ELSIF Device.bFirstCycle THEN
	(* first call of the server device since reboot/reset *)
	bReady := FALSE;
	_PresentValue_Priority12 := BACnetBinaryPV_NULL;
ELSE
	(* server device not ready, reset local ready also *)
	bReady := FALSE;
	nErrorId := nERR_OPERATIONAL;
END_IF
(* set error flag *)
bError := (nErrorId <> nERR_NO_ERROR);
END_FUNCTION_BLOCK

(* POU FB_BACnet_BinaryOutput_ADS, ST *)
FUNCTION_BLOCK FB_BACnet_BinaryOutput_ADS
VAR_INPUT
	bEnablePV		: BOOL;
	bPV				: BOOL; (* present value bool type *)
	bManual			: BOOL; (* FALSE --> TRUE: write present_value immediately, FALSE: only write present_value on-change, TRUE: write present_value on-change and when device turns operational *)
	ePriority		: E_BACNETPRIORITY := BACNETPRIORITY_12;
END_VAR
VAR_IN_OUT
	Device			: FB_BACnet_Device;
END_VAR
VAR_OUTPUT
	bReady			: BOOL;
	bPvDone			: BOOL; (* present_value written over ADS *)
	bPresentValue	: BOOL;
	bOverridden		: BOOL;
	bOutOfService	: BOOL;
	bFault			: BOOL;
	bInAlarm		: BOOL;
	bError			: BOOL;
	nErrorId		: UINT;
	nAdsErrorId		: UDINT;
END_VAR
VAR
	_PresentValue AT%I*: WORD; 			(* ~(BACnet_PresentValue 			:		: )
								   			(BACnet_ObjectType 				: BO	: )	*)
    _PresentValue_Ads : WORD;
	_StatusFlags AT%I*: WORD; 			(* ~(BACnet_StatusFlags 			:		: )	*)
	_ObjectId AT%I*: DWORD;				(* ~(BACnet_ObjectIdentifier			 :		: LINK) *)
	_StatusFlagsBits : ST_BACnet_StatusFlags;
	_nUpdateCount : UDINT := 0;
	_WriteProp : FB_BACnet_WriteProp;
	_rtrigManual : R_TRIG;
	_bEnPvOld : BOOL;
	_nObjType : E_BACNETOBJECTTYPE;
END_VAR
VAR CONSTANT
	nERR_NO_ERROR		: UINT := 0;
	nERR_WRONG_MAPPING	: UINT := 2;
	nERR_OPERATIONAL	: UINT := 3;
	nERR_WRONG_TYPE		: UINT := 4;
END_VAR
(* update server device *)
IF Device._nUpdateCount = _nUpdateCount THEN
	Device();
END_IF
(* remind current number of update counter *)
_nUpdateCount := Device._nUpdateCount;

(* trigger on manual flag *)
_rtrigManual(CLK:= bManual, Q=> );

(* decode object type *)
_nObjType := F_BACnet_GetObjType(_ObjectId);

(* check BitString format of StatusFlags --> if StatusFlags are less than 4, object isn't linked correctly *)
IF _nObjType <> BACnetObjectType_BinaryOutput THEN
	(* wrong mapped object type *)
	nErrorId := nERR_WRONG_TYPE;
	bReady := FALSE;
	bPvDone := FALSE;

ELSIF (_StatusFlags < 4) THEN
	(* wrong mapping *)
	nErrorId := nERR_WRONG_MAPPING;
	bReady := FALSE;
	bPvDone := FALSE;

ELSIF Device.bOperational THEN
	(* write present_value on manual trigger, on-change and on operational recover *)
	IF		_rtrigManual.Q
		OR	((F_BACnet_IsFinite(_PresentValue_Ads) <> F_BACnet_IsFinite(_PresentValue_Ads)) AND bEnablePV)
		OR	(bPV <> F_BinPV_To_Bool(_PresentValue_Ads) AND bEnablePV)
		OR	((NOT bReady) AND bManual)
		OR	(bEnablePV <> _bEnPvOld)
	THEN
		_WriteProp.bExecute := TRUE;
		bPvDone := FALSE;
		(* write depending on enable state *)
		_PresentValue_Ads := F_Bool_To_BinPV(bEnablePV, bPV);
		_bEnPvOld := bEnablePV;
	END_IF

	(* ready state *)
	bReady := TRUE;
	nErrorId := nERR_NO_ERROR;


	(* present value *)
	bPresentValue := F_BinPV_To_Bool(_PresentValue);

	(* build bit states *)
	_StatusFlagsBits := F_BACnet_StatusFlags(_StatusFlags);

	(* copy states to output *)
	bOverridden := _StatusFlagsBits.overridden;
	bOutOfService := _StatusFlagsBits.out_of_service;
	bFault := _StatusFlagsBits.fault;
	bInAlarm := _StatusFlagsBits.in_alarm;

ELSIF Device.bFirstCycle THEN
	(* first call of the server device since reboot/reset *)
	bReady := FALSE;
	bPvDone := FALSE;
ELSE
	(* server device not ready, reset local ready also *)
	bReady := FALSE;
	nErrorId := nERR_OPERATIONAL;
	bPvDone := FALSE;
END_IF

(* call write property command *)
_WriteProp(
	BACnetDevicePort	:= Device.nAdsPort,
	bExecute			:= ,
	sNetId				:= Device.sAmsNetId,
	ObjectType			:= _nObjType,
	PropertyID			:= BACnetPropertyIdentifier_PresentValue,
	Priority			:= ePriority,
	DataType			:= BACnetDataType_BinaryPV,
	ObjectInstance		:= F_BACnet_GetObjInstance(_ObjectId),
	ptrValue			:= ADR(_PresentValue_Ads),
	nLenValue			:= SIZEOF(_PresentValue_Ads),
	bDone				=> ,
	bBusy				=> ,
	bError				=> ,
	nErrID				=> nAdsErrorId);

(* set done flag *)
IF _WriteProp.bExecute AND (NOT _WriteProp.bBusy) THEN
	(* reset execution bit *)
	_WriteProp(bExecute := FALSE);
	(* check if command was finished with error *)
	IF _WriteProp.bError THEN
		IF bManual THEN
			(* retrigger if manual flag is set *)
			_WriteProp.bExecute := TRUE;
		END_IF
		bPvDone := FALSE;
	ELSE
		(* successful written *)
		bPvDone	:= TRUE;
	END_IF
END_IF

(* set error flag *)
bError := (nErrorId <> nERR_NO_ERROR) OR (nAdsErrorId <> 0);
END_FUNCTION_BLOCK

(* POU FB_BACnet_BinaryOutput_EX, ST *)
FUNCTION_BLOCK FB_BACnet_BinaryOutput_EX
VAR_INPUT
	bEnablePV	: BOOL; (* enable present value with priority x in priority array, FALSE = priority x disable (NULL) *)
	bPV			: BOOL; (* present value bool type *)
END_VAR
VAR_IN_OUT
	Device		: FB_BACnet_Device;
END_VAR
VAR_OUTPUT
	bReady			: BOOL;
	bPresentValue	: BOOL;
	bOverridden		: BOOL;
	bOutOfService	: BOOL;
	bFault			: BOOL;
	bInAlarm		: BOOL;
	bNoOutput		: BOOL;
	bOpenLoop		: BOOL;
	bShortedLoop	: BOOL;
	bOtherFault		: BOOL;
	eEventState		: E_BACNETEVENTSTATE;
	bAckedTrans_ToOffNormal : BOOL;
	bAckedTrans_ToFault		: BOOL;
	bAckedTrans_ToNormal	: BOOL;
	nActivePrio		: UINT;
	bError			: BOOL;
	nErrorId		: UINT;
END_VAR
VAR_INPUT
END_VAR
VAR
	_PresentValue AT%I*: WORD; 			(* ~(BACnet_PresentValue 			:		: )
								   			(BACnet_ObjectType 				: BO	: )	*)
    _PresentValue_Priority12 AT%Q*: WORD;(* ~(BACnet_PresentValue_Priority12	:		: )	*)
	_StatusFlags AT%I*: WORD; 			(* ~(BACnet_StatusFlags 			:		: )	*)
	_StatusFlagsBits : ST_BACnet_StatusFlags;
	_EventState AT%I*: WORD; 			(* ~(BACnet_EventState 				:		: )	*)
	_Reliability AT%I*: WORD;			(* ~(BACnet_Reliability 			:		: )	*)
	_ActivePriority AT%I*: UDINT; 		(* ~(BACnet_ActivePriority 			:		: )	*)
	_AckedTransitions AT%I*:WORD;	(* ~(BACnet_AckedTransitions:		: ) *)
	_AckedTransBits : ST_BACnet_EventTransitionBits;
	_nUpdateCount : UDINT := 0;
END_VAR
VAR CONSTANT
	nERR_NO_ERROR		: UINT := 0;
	nERR_WRONG_MAPPING	: UINT := 2;
	nERR_OPERATIONAL	: UINT := 3;
END_VAR
(* update server device *)
IF Device._nUpdateCount = _nUpdateCount THEN
	Device();
END_IF
(* remind current number of update counter *)
_nUpdateCount := Device._nUpdateCount;

(* check BitString format of StatusFlags --> if StatusFlags are less than 4, object isn't linked correctly *)
IF (_StatusFlags < 4) OR _AckedTransitions < 5 THEN
	(* wrong mapping *)
	nErrorId := nERR_WRONG_MAPPING;
	bReady := FALSE;

ELSIF Device.bOperational THEN
	(* ready state *)
	bReady := TRUE;
	nErrorId := nERR_NO_ERROR;

	(* write into priority array *)
	_PresentValue_Priority12 := F_Bool_To_BinPV(bEnablePV, bPV);

	(* present value *)
	bPresentValue := F_BinPV_To_Bool(_PresentValue);

	(* build bit states *)
	_StatusFlagsBits := F_BACnet_StatusFlags(_StatusFlags);
	_AckedTransBits		:= F_BACnet_EventTransitionFlags(_AckedTransitions);

	(* copy states to output *)
	bOverridden := _StatusFlagsBits.overridden;
	bOutOfService := _StatusFlagsBits.out_of_service;
	bFault := _StatusFlagsBits.fault;
	bInAlarm := _StatusFlagsBits.in_alarm;
	bNoOutput := (_Reliability = BACnetReliability_no_output);
	bOpenLoop := (_Reliability = BACnetReliability_open_loop);
	bShortedLoop := (_Reliability = BACnetReliability_shorted_loop);
	bOtherFault := (_Reliability = BACnetReliability_unreliable_other);
	bAckedTrans_ToOffNormal := _AckedTransBits.to_offnormal;
	bAckedTrans_ToFault := _AckedTransBits.to_fault;
	bAckedTrans_ToNormal := _AckedTransBits.to_normal;

	(* convert enumeration *)
	eEventState := _EventState;

	(* copy active priority *)
	nActivePrio := UDINT_TO_UINT(_ActivePriority);
ELSIF Device.bFirstCycle THEN
	(* first call of the server device since reboot/reset *)
	bReady := FALSE;
	_PresentValue_Priority12 := BACnetBinaryPV_NULL;
ELSE
	(* server device not ready, reset local ready also *)
	bReady := FALSE;
	nErrorId := nERR_OPERATIONAL;
END_IF
(* set error flag *)
bError := (nErrorId <> nERR_NO_ERROR);
END_FUNCTION_BLOCK

(* POU FB_BACnet_BinaryOutput_RAW, ST *)
FUNCTION_BLOCK FB_BACnet_BinaryOutput_RAW
VAR_INPUT
	bEnablePV	: BOOL; (* enable present value with priority x in priority array, FALSE = priority x disable (NULL) *)
	bPV			: BOOL; (* present value bool type *)
END_VAR
VAR_IN_OUT
	Device		: FB_BACnet_Device;
END_VAR
VAR_OUTPUT
	bReady			: BOOL;
	bPresentValue	: BOOL;
	bOverridden		: BOOL;
	bOutOfService	: BOOL;
	bFault			: BOOL;
	bInAlarm		: BOOL;
	bAckedTrans_ToOffNormal : BOOL;
	bAckedTrans_ToFault		: BOOL;
	bAckedTrans_ToNormal	: BOOL;
	bError			: BOOL;
	nErrorId		: UINT;
	bRawOut			AT%I*: BOOL;(* ~(BACnet_RawIoBinaryBoolValue : : ) *)
END_VAR
VAR
	_PresentValue AT%I*: WORD; 			(* ~(BACnet_PresentValue 			:		: )
								   			(BACnet_ObjectType 				: BO	: )	*)
    _PresentValue_Priority12 AT%Q*: WORD;(* ~(BACnet_PresentValue_Priority12	:		: )	*)
	_StatusFlags AT%I*: WORD; 			(* ~(BACnet_StatusFlags 			:		: )	*)
	_AckedTransitions AT%I*:WORD;		(* ~(BACnet_AckedTransitions:		: ) *)
	_AckedTransBits : ST_BACnet_EventTransitionBits;
	_StatusFlagsBits : ST_BACnet_StatusFlags;
	_nUpdateCount : UDINT := 0;
END_VAR
VAR CONSTANT
	nERR_NO_ERROR		: UINT := 0;
	nERR_WRONG_MAPPING	: UINT := 2;
	nERR_OPERATIONAL	: UINT := 3;
END_VAR
(* update server device *)
IF Device._nUpdateCount = _nUpdateCount THEN
	Device();
END_IF
(* remind current number of update counter *)
_nUpdateCount := Device._nUpdateCount;

(* check BitString format of StatusFlags --> if StatusFlags are less than 4, object isn't linked correctly *)
IF (_StatusFlags < 4) OR _AckedTransitions < 5 THEN
	(* wrong mapping *)
	nErrorId := nERR_WRONG_MAPPING;
	bReady := FALSE;

ELSIF Device.bOperational THEN
	(* ready state *)
	bReady := TRUE;
	nErrorId := nERR_NO_ERROR;

	(* write into priority array *)
	_PresentValue_Priority12 := F_Bool_To_BinPV(bEnablePV, bPV);

	(* present value *)
	bPresentValue := F_BinPV_To_Bool(_PresentValue);

	(* build bit states *)
	_StatusFlagsBits := F_BACnet_StatusFlags(_StatusFlags);
	_AckedTransBits		:= F_BACnet_EventTransitionFlags(_AckedTransitions);

	(* copy states to output *)
	bOverridden := _StatusFlagsBits.overridden;
	bOutOfService := _StatusFlagsBits.out_of_service;
	bFault := _StatusFlagsBits.fault;
	bInAlarm := _StatusFlagsBits.in_alarm;
	bAckedTrans_ToOffNormal := _AckedTransBits.to_offnormal;
	bAckedTrans_ToFault := _AckedTransBits.to_fault;
	bAckedTrans_ToNormal := _AckedTransBits.to_normal;

ELSIF Device.bFirstCycle THEN
	(* first call of the server device since reboot/reset *)
	bReady := FALSE;
	_PresentValue_Priority12 := BACnetBinaryPV_NULL;
ELSE
	(* server device not ready, reset local ready also *)
	bReady := FALSE;
	nErrorId := nERR_OPERATIONAL;
END_IF
(* set error flag *)
bError := (nErrorId <> nERR_NO_ERROR);
END_FUNCTION_BLOCK

(* POU FB_BACnet_BinaryValue, ST *)
FUNCTION_BLOCK FB_BACnet_BinaryValue
VAR_INPUT
	bEnablePV	: BOOL; (* enable present value with priority x in priority array, FALSE = priority x disable (NULL) *)
	bPV			: BOOL; (* present value bool type *)
END_VAR
VAR_IN_OUT
	Device		: FB_BACnet_Device;
END_VAR
VAR_OUTPUT
	bReady			: BOOL;
	bPresentValue	: BOOL;
	bOverridden		: BOOL;
	bOutOfService	: BOOL;
	bFault			: BOOL;
	bInAlarm		: BOOL;
	bError			: BOOL;
	nErrorId		: UINT;
END_VAR
VAR
	_PresentValue AT%I*: WORD; 			(* ~(BACnet_PresentValue 			:		: )
								   			(BACnet_ObjectType 				: BV	: )	*)
    _PresentValue_Priority12 AT%Q*: WORD;(* ~(BACnet_PresentValue_Priority12	:		: )	*)
	_StatusFlags AT%I*: WORD; 			(* ~(BACnet_StatusFlags 			:		: )	*)
	_StatusFlagsBits : ST_BACnet_StatusFlags;
	_nUpdateCount : UDINT := 0;
END_VAR
VAR CONSTANT
	nERR_NO_ERROR		: UINT := 0;
	nERR_WRONG_MAPPING	: UINT := 2;
	nERR_OPERATIONAL	: UINT := 3;
END_VAR
(* update server device *)
IF Device._nUpdateCount = _nUpdateCount THEN
	Device();
END_IF
(* remind current number of update counter *)
_nUpdateCount := Device._nUpdateCount;

(* check BitString format of StatusFlags --> if StatusFlags are less than 4, object isn't linked correctly *)
IF (_StatusFlags < 4) THEN
	(* wrong mapping *)
	nErrorId := nERR_WRONG_MAPPING;
	bReady := FALSE;

ELSIF Device.bOperational THEN
	(* ready state *)
	bReady := TRUE;
	nErrorId := nERR_NO_ERROR;

	(* write into priority array *)
	_PresentValue_Priority12 := F_Bool_To_BinPV(bEnablePV, bPV);

	(* present value *)
	bPresentValue := F_BinPV_To_Bool(_PresentValue);

	(* build bit states *)
	_StatusFlagsBits := F_BACnet_StatusFlags(_StatusFlags);

	(* copy states to output *)
	bOverridden := _StatusFlagsBits.overridden;
	bOutOfService := _StatusFlagsBits.out_of_service;
	bFault := _StatusFlagsBits.fault;
	bInAlarm := _StatusFlagsBits.in_alarm;

ELSIF Device.bFirstCycle THEN
	(* first call of the server device since reboot/reset *)
	bReady := FALSE;
	_PresentValue_Priority12 := BACnetBinaryPV_NULL;
ELSE
	(* server device not ready, reset local ready also *)
	bReady := FALSE;
	nErrorId := nERR_OPERATIONAL;
END_IF
(* set error flag *)
bError := (nErrorId <> nERR_NO_ERROR);
END_FUNCTION_BLOCK

(* POU FB_BACnet_BinaryValue_ADS, ST *)
FUNCTION_BLOCK FB_BACnet_BinaryValue_ADS
VAR_INPUT
	bEnablePV		: BOOL;
	bPV				: BOOL; (* present value bool type *)
	bManual			: BOOL; (* FALSE --> TRUE: write present_value immediately, FALSE: only write present_value on-change, TRUE: write present_value on-change and when device turns operational *)
	ePriority		: E_BACNETPRIORITY := BACNETPRIORITY_12;
END_VAR
VAR_IN_OUT
	Device			: FB_BACnet_Device;
END_VAR
VAR_OUTPUT
	bReady			: BOOL;
	bPvDone			: BOOL; (* present_value written over ADS *)
	bPresentValue	: BOOL;
	bOverridden		: BOOL;
	bOutOfService	: BOOL;
	bFault			: BOOL;
	bInAlarm		: BOOL;
	bError			: BOOL;
	nErrorId		: UINT;
	nAdsErrorId		: UDINT;
END_VAR
VAR
	_PresentValue AT%I*: WORD; 			(* ~(BACnet_PresentValue 			:		: )
								   			(BACnet_ObjectType 				: BV	: )	*)
    _PresentValue_Ads : WORD;
	_StatusFlags AT%I*: WORD; 			(* ~(BACnet_StatusFlags 			:		: )	*)
	_ObjectId AT%I*: DWORD;				(* ~(BACnet_ObjectIdentifier			 :		: LINK) *)
	_StatusFlagsBits : ST_BACnet_StatusFlags;
	_nUpdateCount : UDINT := 0;
	_WriteProp : FB_BACnet_WriteProp;
	_rtrigManual : R_TRIG;
	_bEnPvOld : BOOL;
	_nObjType : E_BACNETOBJECTTYPE;
END_VAR
VAR CONSTANT
	nERR_NO_ERROR		: UINT := 0;
	nERR_WRONG_MAPPING	: UINT := 2;
	nERR_OPERATIONAL	: UINT := 3;
	nERR_WRONG_TYPE		: UINT := 4;
END_VAR
(* update server device *)
IF Device._nUpdateCount = _nUpdateCount THEN
	Device();
END_IF
(* remind current number of update counter *)
_nUpdateCount := Device._nUpdateCount;

(* trigger on manual flag *)
_rtrigManual(CLK:= bManual, Q=> );

(* decode object type *)
_nObjType := F_BACnet_GetObjType(_ObjectId);

(* check BitString format of StatusFlags --> if StatusFlags are less than 4, object isn't linked correctly *)
IF _nObjType <> BACnetObjectType_BinaryValue THEN
	(* wrong mapped object type *)
	nErrorId := nERR_WRONG_TYPE;
	bReady := FALSE;
	bPvDone := FALSE;

ELSIF (_StatusFlags < 4) THEN
	(* wrong mapping *)
	nErrorId := nERR_WRONG_MAPPING;
	bReady := FALSE;
	bPvDone := FALSE;

ELSIF Device.bOperational THEN
	(* write present_value on manual trigger, on-change and on operational recover *)
	IF		_rtrigManual.Q
		OR	((F_BACnet_IsFinite(_PresentValue_Ads) <> F_BACnet_IsFinite(_PresentValue_Ads)) AND bEnablePV)
		OR	(bPV <> F_BinPV_To_Bool(_PresentValue_Ads) AND bEnablePV)
		OR	((NOT bReady) AND bManual)
		OR	(bEnablePV <> _bEnPvOld)
	THEN
		_WriteProp.bExecute := TRUE;
		bPvDone := FALSE;
		(* write depending on enable state *)
		_PresentValue_Ads := F_Bool_To_BinPV(bEnablePV, bPV);
		_bEnPvOld := bEnablePV;
	END_IF

	(* ready state *)
	bReady := TRUE;
	nErrorId := nERR_NO_ERROR;

	(* present value *)
	bPresentValue := F_BinPV_To_Bool(_PresentValue);

	(* build bit states *)
	_StatusFlagsBits := F_BACnet_StatusFlags(_StatusFlags);

	(* copy states to output *)
	bOverridden := _StatusFlagsBits.overridden;
	bOutOfService := _StatusFlagsBits.out_of_service;
	bFault := _StatusFlagsBits.fault;
	bInAlarm := _StatusFlagsBits.in_alarm;

ELSIF Device.bFirstCycle THEN
	(* first call of the server device since reboot/reset *)
	bReady := FALSE;
	bPvDone := FALSE;
ELSE
	(* server device not ready, reset local ready also *)
	bReady := FALSE;
	nErrorId := nERR_OPERATIONAL;
	bPvDone := FALSE;
END_IF

(* call write property command *)
_WriteProp(
	BACnetDevicePort	:= Device.nAdsPort,
	bExecute			:= ,
	sNetId				:= Device.sAmsNetId,
	ObjectType			:= _nObjType,
	PropertyID			:= BACnetPropertyIdentifier_PresentValue,
	Priority			:= ePriority,
	DataType			:= BACnetDataType_BinaryPV,
	ObjectInstance		:= F_BACnet_GetObjInstance(_ObjectId),
	ptrValue			:= ADR(_PresentValue_Ads),
	nLenValue			:= SIZEOF(_PresentValue_Ads),
	bDone				=> ,
	bBusy				=> ,
	bError				=> ,
	nErrID				=> nAdsErrorId);

(* set done flag *)
IF _WriteProp.bExecute AND (NOT _WriteProp.bBusy) THEN
	(* reset execution bit *)
	_WriteProp(bExecute := FALSE);
	(* check if command was finished with error *)
	IF _WriteProp.bError THEN
		IF bManual THEN
			(* retrigger if manual flag is set *)
			_WriteProp.bExecute := TRUE;
		END_IF
		bPvDone := FALSE;
	ELSE
		(* successful written *)
		bPvDone	:= TRUE;
	END_IF
END_IF

(* set error flag *)
bError := (nErrorId <> nERR_NO_ERROR) OR (nAdsErrorId <> 0);
END_FUNCTION_BLOCK

(* POU FB_BACnet_BinaryValue_EX, ST *)
FUNCTION_BLOCK FB_BACnet_BinaryValue_EX
VAR_INPUT
	bEnablePV	: BOOL; (* enable present value with priority x in priority array, FALSE = priority x disable (NULL) *)
	bPV			: BOOL; (* present value bool type *)
END_VAR
VAR_IN_OUT
	Device		: FB_BACnet_Device;
END_VAR
VAR_OUTPUT
	bReady			: BOOL;
	bPresentValue	: BOOL;
	bOverridden		: BOOL;
	bOutOfService	: BOOL;
	bFault			: BOOL;
	bInAlarm		: BOOL;
	bOtherFault		: BOOL;
	eEventState		: E_BACNETEVENTSTATE;
	bAckedTrans_ToOffNormal : BOOL;
	bAckedTrans_ToFault		: BOOL;
	bAckedTrans_ToNormal	: BOOL;
	nActivePrio		: UINT;
	bError			: BOOL;
	nErrorId		: UINT;
END_VAR
VAR

	_PresentValue AT%I*: WORD; 			(* ~(BACnet_PresentValue 			:		: )
								   			(BACnet_ObjectType 				: BV	: )	*)
    _PresentValue_Priority12 AT%Q*: WORD;(* ~(BACnet_PresentValue_Priority12	:		: )	*)
	_StatusFlags AT%I*: WORD; 			(* ~(BACnet_StatusFlags 			:		: )	*)
	_StatusFlagsBits : ST_BACnet_StatusFlags;
	_EventState AT%I*: WORD; 			(* ~(BACnet_EventState 				:		: )	*)
	_Reliability AT%I*: WORD;			(* ~(BACnet_Reliability 			:		: )	*)
	_ActivePriority AT%I*: UDINT; 		(* ~(BACnet_ActivePriority 			:		: )	*)
	_AckedTransitions AT%I*:WORD;		(* ~(BACnet_AckedTransitions:		: ) *)
	_AckedTransBits : ST_BACnet_EventTransitionBits;
	_nUpdateCount : UDINT := 0;
END_VAR
VAR CONSTANT
	nERR_NO_ERROR		: UINT := 0;
	nERR_WRONG_MAPPING	: UINT := 2;
	nERR_OPERATIONAL	: UINT := 3;
END_VAR
(* update server device *)
IF Device._nUpdateCount = _nUpdateCount THEN
	Device();
END_IF
(* remind current number of update counter *)
_nUpdateCount := Device._nUpdateCount;

(* check BitString format of StatusFlags --> if StatusFlags are less than 4, object isn't linked correctly *)
IF (_StatusFlags < 4) OR _AckedTransitions < 5 THEN
	(* wrong mapping *)
	nErrorId := nERR_WRONG_MAPPING;
	bReady := FALSE;

ELSIF Device.bOperational THEN
	(* ready state *)
	bReady := TRUE;
	nErrorId := nERR_NO_ERROR;

	(* write into priority array *)
	_PresentValue_Priority12 := F_Bool_To_BinPV(bEnablePV, bPV);

	(* present value *)
	bPresentValue := F_BinPV_To_Bool(_PresentValue);

	(* build bit states *)
	_StatusFlagsBits := F_BACnet_StatusFlags(_StatusFlags);
	_AckedTransBits		:= F_BACnet_EventTransitionFlags(_AckedTransitions);

	(* copy states to output *)
	bOverridden := _StatusFlagsBits.overridden;
	bOutOfService := _StatusFlagsBits.out_of_service;
	bFault := _StatusFlagsBits.fault;
	bInAlarm := _StatusFlagsBits.in_alarm;
	bOtherFault := (_Reliability = BACnetReliability_unreliable_other);
	bAckedTrans_ToOffNormal := _AckedTransBits.to_offnormal;
	bAckedTrans_ToFault := _AckedTransBits.to_fault;
	bAckedTrans_ToNormal := _AckedTransBits.to_normal;

	(* convert enumeration *)
	eEventState := _EventState;

	(* copy active priority *)
	nActivePrio := UDINT_TO_UINT(_ActivePriority);
ELSIF Device.bFirstCycle THEN
	(* first call of the server device since reboot/reset *)
	bReady := FALSE;
	_PresentValue_Priority12 := BACnetBinaryPV_NULL;
ELSE
	(* server device not ready, reset local ready also *)
	bReady := FALSE;
	nErrorId := nERR_OPERATIONAL;
END_IF
(* set error flag *)
bError := (nErrorId <> nERR_NO_ERROR);
END_FUNCTION_BLOCK

(* POU FB_BACnet_Calendar, ST *)
FUNCTION_BLOCK FB_BACnet_Calendar
VAR_IN_OUT
	Device	: FB_BACnet_Device;
END_VAR
VAR_OUTPUT
	bReady			: BOOL;
	bPresentValue	: BOOL;
	bError			: BOOL;
	nErrorId		: UINT;
END_VAR
VAR
	_PresentValue AT%I*: BOOL;	(* ~(BACnet_PresentValue 				 :		: )
									(BACnet_ObjectType 					 : CAL	: )	*)
	_nUpdateCount : UDINT := 0;
END_VAR
VAR CONSTANT
	nERR_NO_ERROR		: UINT := 0;
	nERR_OPERATIONAL	: UINT := 3;
END_VAR
(* update server device *)
IF Device._nUpdateCount = _nUpdateCount THEN
	Device();
END_IF
(* remind current number of update counter *)
_nUpdateCount := Device._nUpdateCount;

IF Device.bOperational THEN
	(* ready state *)
	bReady := TRUE;
	nErrorId := nERR_NO_ERROR;
	(* present value *)
	bPresentValue := _PresentValue;
ELSE
	(* server device not ready, reset local ready also *)
	bReady := FALSE;
	nErrorId := nERR_OPERATIONAL;
END_IF
(* set error flag *)
bError := (nErrorId <> nERR_NO_ERROR);
END_FUNCTION_BLOCK

(* POU FB_BACnet_Command, ST *)
FUNCTION_BLOCK FB_BACnet_Command
VAR_INPUT
	bEnablePV		: BOOL;
	nPV				: UDINT;
	bRetrigger		: BOOL; (* execute selected action on raising edge again *)
END_VAR
VAR_IN_OUT
	Device	: FB_BACnet_Device;
END_VAR
VAR_OUTPUT
	bReady			: BOOL;
	nPresentValue	: UDINT;
	bAllWritesOk	: BOOL; (* all actions in selected action list are written *)
	bInProcess		: BOOL; (* object is busy *)
	bError			: BOOL;
	nErrorId		: UINT;
END_VAR
VAR
	_PresentValueIn AT%I*: UDINT; 		(* ~(BACnet_PresentValue 				 :		: )
								   			(BACnet_ObjectType 					 : CMD	: )	*)
	_InProcess AT%I*: BOOL;				(* ~(BACnet_InProcess 					 :		: )	*)
	_AllWritesSuccessful AT%I*: BOOL;	(* ~(BACnet_AllWritesSuccessful			 :		: )	*)
    _PresentValueOut AT%Q*: UDINT;		(* ~(BACnet_PresentValue	 	   		 :      : )	*)
	_nUpdateCount : UDINT := 0;
	_rtrigRetriggerPv : R_TRIG;
END_VAR
VAR CONSTANT
	nERR_NO_ERROR		: UINT := 0;
	nERR_OPERATIONAL	: UINT := 3;
END_VAR
(* update server device *)
IF Device._nUpdateCount = _nUpdateCount THEN
	Device();
END_IF
(* remind current number of update counter *)
_nUpdateCount := Device._nUpdateCount;

(* call trigger *)
_rtrigRetriggerPv(CLK:= bRetrigger, Q=> );

IF Device.bOperational THEN
	(* ready state *)
	bReady := TRUE;
	nErrorId := nERR_NO_ERROR;
	(* present value from BACnet *)
	nPresentValue := _PresentValueIn;
	(* present value to BACnet *)
	IF bEnablePV THEN
		IF _rtrigRetriggerPv.Q THEN
			(* trigger action list *)
			_PresentValueOut := 0;
		ELSE
			(* set present value *)
			_PresentValueOut := nPV;
		END_IF
	ELSE
		(* deactivate mapped present value --> other objects can write to property *)
		_PresentValueOut := 16#FFFFFFFF;
	END_IF
	(* other states *)
	bAllWritesOk := _AllWritesSuccessful;
	bInProcess := _InProcess;
ELSIF Device.bFirstCycle THEN
	(* first call of the server device since reboot/reset *)
	bReady := FALSE;
	_PresentValueOut := 0;
ELSE
	(* server device not ready, reset local ready also *)
	bReady := FALSE;
	nErrorId := nERR_OPERATIONAL;
END_IF
(* set error flag *)
bError := (nErrorId <> nERR_NO_ERROR);
END_FUNCTION_BLOCK

(* POU FB_BACnet_File, ST *)
FUNCTION_BLOCK FB_BACnet_File
VAR_IN_OUT
	Device	: FB_BACnet_Device;
END_VAR
VAR_OUTPUT
	bReady			: BOOL;
	nFileSize		: UDINT;
	bError			: BOOL;
	nErrorId		: UINT;
END_VAR
VAR
	_FileSize 			AT%I*: UDINT; 	(* ~(BACnet_FileSize 					 :		: )
					   						(BACnet_ObjectType 					 : FILE	: )	*)
	_nUpdateCount		: UDINT := 0;
END_VAR
VAR CONSTANT
	nERR_NO_ERROR		: UINT := 0;
	nERR_OPERATIONAL	: UINT := 3;
END_VAR
(* update server device *)
IF Device._nUpdateCount = _nUpdateCount THEN
	Device();
END_IF
(* remind current number of update counter *)
_nUpdateCount := Device._nUpdateCount;

IF Device.bOperational THEN
	(* ready state *)
	bReady := TRUE;
	nErrorId := nERR_NO_ERROR;
	nFileSize := _FileSize;
ELSE
	(* server device not ready, reset local ready also *)
	bReady := FALSE;
	nErrorId := nERR_OPERATIONAL;
END_IF
(* set error flag *)
bError := (nErrorId <> nERR_NO_ERROR);
END_FUNCTION_BLOCK

(* POU FB_BACnet_GetDiagInfo, ST *)
FUNCTION_BLOCK FB_BACnet_GetDiagInfo
VAR_INPUT
	sNetId		: T_AmsNetId;
	bExecute	: BOOL;
	tTimeout	: TIME := tBACnet_ADSTimeOut;
END_VAR
VAR_OUTPUT
	bBusy		: BOOL;
	bError		: BOOL;
	nErrID		: UDINT;
	stInfo		: ST_BACnet_Diagnosis;
END_VAR
VAR
	_fbAdsRead	: ADSREAD;
END_VAR
(* call ADS read function to receive info data *)
_fbAdsRead(
	NETID	:= sNetId,
	PORT	:= 16#FFFF, (* ADS port of BACnet device adapter *)
	IDXGRP	:= 16#8000000F,
	IDXOFFS	:= 16#0000,
	LEN		:= SIZEOF(stInfo),
	DESTADDR:= ADR(stInfo),
	READ	:= bExecute,
	TMOUT	:= tTimeout,
	BUSY	=> bBusy,
	ERR		=> bError,
	ERRID	=> nErrID);
END_FUNCTION_BLOCK

(* POU FB_BACnet_Group, ST *)
FUNCTION_BLOCK FB_BACnet_Group
VAR_IN_OUT
	Device	: FB_BACnet_Device;
END_VAR
VAR_OUTPUT
	bReady			: BOOL;
	bError			: BOOL;
	nErrorId		: UINT;
END_VAR
VAR
	_ObjectType: E_BACNETOBJECTTYPE;	(* ~ (BACNET_OBJECTTYPE : GROUP : )	*)
	_nUpdateCount : UDINT := 0;
END_VAR
VAR CONSTANT
	nERR_NO_ERROR		: UINT := 0;
	nERR_OPERATIONAL	: UINT := 3;
END_VAR
_ObjectType := BACnetObjectType_Group;
(* update server device *)
IF Device._nUpdateCount = _nUpdateCount THEN
	Device();
END_IF
(* remind current number of update counter *)
_nUpdateCount := Device._nUpdateCount;

IF Device.bOperational THEN
	(* ready state *)
	bReady := TRUE;
	nErrorId := nERR_NO_ERROR;
ELSE
	(* server device not ready, reset local ready also *)
	bReady := FALSE;
	nErrorId := nERR_OPERATIONAL;
END_IF
(* set error flag *)
bError := (nErrorId <> nERR_NO_ERROR);
END_FUNCTION_BLOCK

(* POU FB_BACnet_Loop, ST *)
FUNCTION_BLOCK FB_BACnet_Loop
VAR_INPUT
	bEnable			: BOOL; (* enable LOOP object (false = out_of_service) *)
END_VAR
VAR_IN_OUT
	Device	: FB_BACnet_Device;
END_VAR
VAR_OUTPUT
	bReady			: BOOL;
	fSetPoint		: REAL;
	fControlledValue: REAL;
	fPresentValue	: REAL;
	fPropBand		: REAL; (* controller output in range of -100...100% in relation to Min.-/Max.-output *)
	bOverridden		: BOOL;
	bOutOfService	: BOOL;
	bFault			: BOOL;
	bInAlarm		: BOOL;
	bOpenLoop		: BOOL;
	bOtherFault		: BOOL;
	bError			: BOOL;
	nErrorId		: UINT;
END_VAR
VAR
	_ControlledVariableValue AT%I*: REAL;	(* ~ (BACnet_ControlledVariableValue 		:		: )
												 (BACnet_ObjectType						: LOOP	: )	*)
	_Setpoint AT%I*:REAL;					(* ~ (BACnet_Setpoint				 		:		: )	*)
	_ProportionalConstant AT%I*:REAL;		(* ~ (BACnet_ProportionalConstant	 		:		: )	*)
	_IntegralConstant AT%I*:REAL;			(* ~ (BACnet_IntegralConstant	 			:		: )	*)
	_DerivativeConstant AT%I*:REAL;			(* ~ (BACnet_DerivativeConstant	 			:		: )	*)
	_MaximumOutput AT%I*:REAL;				(* ~ (BACnet_MaximumOutput				 	:		: )	*)
	_MinimumOutput AT%I*:REAL;				(* ~ (BACnet_MinimumOutput				 	:		: )	*)
	_Bias AT%I*:REAL;						(* ~ (BACnet_Bias					 		:		: )	*)
	_Reliability AT%I*: E_BACNETRELIABILITY;(* ~ (BACNET_RELIABILITY 					:		: )	*)
	_StatusFlags AT%I*: WORD; 				(* ~ (BACnet_StatusFlags 					: 		: )	*)
	_StatusFlagsBits : ST_BACnet_StatusFlags;
	_ControlAction AT%I*:E_BACNETACTION;	(* ~ (BACNET_ACTION				 			:		: )	*)
	_PresentValueI AT%I*: REAL; 			(* ~ (BACnet_PresentValue 				 	: 		: )	*)
	_PresentValueQ AT%Q*: REAL;				(* ~ (BACnet_PresentValue	 				:		: )	*)
	_OutOfService AT%Q*: BOOL;				(* ~ (BACnet_OutOfService 				 	: 		: )	*)

	_fbGetTaskIndex : GETCURTASKINDEX;
	_rTaskCycleTime : REAL;
	_PidControl : FB_BACnet_PidControl;

	_nUpdateCount : UDINT := 0;
END_VAR
VAR CONSTANT
	nERR_NO_ERROR		: UINT := 0;
	nERR_WRONG_MAPPING	: UINT := 2;
	nERR_OPERATIONAL	: UINT := 3;
END_VAR
(* update server device *)
IF Device._nUpdateCount = _nUpdateCount THEN
	Device();
END_IF
(* remind current number of update counter *)
_nUpdateCount := Device._nUpdateCount;

(* check BitString format of StatusFlags --> if StatusFlags are less than 4, object isn't linked correctly *)
IF (_StatusFlags < 4) THEN
	(* wrong mapping *)
	nErrorId := nERR_WRONG_MAPPING;
	bReady := FALSE;

ELSIF Device.bOperational THEN
	(* ready state *)
	bReady := TRUE;
	nErrorId := nERR_NO_ERROR;

	(* decode status flags *)
	_StatusFlagsBits := F_BACnet_StatusFlags(_StatusFlags);

	(* copy states to output *)
	bOverridden := _StatusFlagsBits.overridden;
	bOutOfService := _StatusFlagsBits.out_of_service;
	bFault := _StatusFlagsBits.fault;
	bInAlarm := _StatusFlagsBits.in_alarm;
	bOpenLoop := (_Reliability = BACnetReliability_open_loop);
	bOtherFault := (_Reliability = BACnetReliability_unreliable_other);

	(* external logic set disable to FALSE *)
	IF (NOT bEnable) THEN
		_PidControl.bReset			:= TRUE;
		_OutOfService				:= TRUE;

	(* check reliability *)
	ELSIF _Reliability <> BACnetReliability_no_fault_detected THEN
		_PidControl.bReset			:= TRUE;
		_OutOfService				:= FALSE;

	(* is set out of service? *)
	ELSIF _StatusFlagsBits.out_of_service THEN
		_PidControl.bReset			:= TRUE;
		_OutOfService				:= FALSE;

	(* decide the control action (direct or reverse) *)
	ELSIF _ControlAction = BACnetAction_direct THEN
		_PidControl.bReset			:= FALSE;
		_PidControl.fPresentValue	:= _ControlledVariableValue;
		_PidControl.fSetpoint		:= _Setpoint;
		_OutOfService				:= FALSE;

	ELSIF _ControlAction = BACnetAction_reverse THEN
		_PidControl.bReset			:= FALSE;
		_PidControl.fPresentValue	:= _Setpoint;
		_PidControl.fSetpoint		:= _ControlledVariableValue;
		_OutOfService				:= FALSE;

	ELSE
		(* unknown action *)
		_PidControl.bReset			:= TRUE;
		_OutOfService				:= TRUE;
	END_IF

	(* get task cycle time *)
	_fbGetTaskIndex();
	_rTaskCycleTime := SystemTaskInfoArr[_fbGetTaskIndex.index].cycleTime / 10000000.0; (* [s] *)

	(* call PID control function block *)
	_PidControl(
		fCtrlCycleTime	:= _rTaskCycleTime,
		fBias			:= _Bias,
		fKp				:= _ProportionalConstant,
		fKi				:= _IntegralConstant,
		fKd				:= _DerivativeConstant,
		fMaxOutput		:= _MaximumOutput,
		fMinOutput		:= _MinimumOutput,
		nErrorStatus	=>
	);
	_PresentValueQ := _PidControl.fY;

	(* calculate proportional band *)
	IF (_MaximumOutput > 0.0) AND (_MinimumOutput >= 0.0) THEN
		fPropBand := ((_PresentValueQ - _MinimumOutput) / (_MaximumOutput - _MinimumOutput)) * 100.0;
	ELSIF (_MaximumOutput <= 0.0) AND (_MinimumOutput < 0.0) THEN
		fPropBand := ((_PresentValueQ - _MaximumOutput) / (_MaximumOutput - _MinimumOutput)) * 100.0;
	ELSIF (_PresentValueQ > 0.0) AND (_MaximumOutput > 0.0) THEN
		fPropBand := (_PresentValueQ / _MaximumOutput) * 100.0;
	ELSIF (_PresentValueQ < 0.0) AND (_MinimumOutput < 0.0) THEN
		fPropBand := (_PresentValueQ / _MinimumOutput) * -100.0;
	ELSE
		fPropBand := 0.0;
	END_IF

	(* set other outputs *)
	fSetPoint := _Setpoint;
	fPresentValue := _PresentValueI;
	fControlledValue := _ControlledVariableValue;
ELSE
	(* server device not ready, reset local ready also *)
	bReady := FALSE;
	nErrorId := nERR_OPERATIONAL;
END_IF
(* set error flag *)
bError := (nErrorId <> nERR_NO_ERROR);
END_FUNCTION_BLOCK

(* POU FB_BACnet_PidControl, ST *)
FUNCTION_BLOCK FB_BACnet_PidControl
VAR_INPUT
	(* controller input  *)
	fSetpoint				: REAL;	(* setpoint value *)
	fPresentValue			: REAL;	(* actual value *)
	(* reset flag *)
	bReset					: BOOL;
	(* controller values *)
	fCtrlCycleTime			: REAL; (* controller cycle time in seconds [s] *)

	fBias					: REAL; (* bias also active when reset is set to 1 *)
	fKp						: REAL;	(* proportional gain Kp	(P) *)
	fKi						: REAL; (* integral gain Ki (I) *)
	fKd						: REAL;	(* derivative gain Kd (D) *)

	(* maximum ratings *)
	fMaxOutput				: REAL;
	fMinOutput				: REAL;
END_VAR
VAR_OUTPUT
	fY						: REAL; (* controller output command *)
	nErrorStatus			: UINT; (* controller error output (0: no error; >0:error) *)
END_VAR
VAR CONSTANT
	nERR_NOERROR			: UINT := 0; (* no error *)
	nERR_INVALIDPARAM		: UINT := 1; (* invalid parameter *)
	nERR_INVALIDCYCLETIME	: UINT := 2; (* invalid cycle time *)
END_VAR
VAR
	(* Internal Variable *)
	_fE						: REAL;
	_fEOld					: REAL;
	_fYp					: REAL;
	_fYi					: REAL;
	_fYd					: REAL;
END_VAR
(* preset error number *)
nErrorStatus	:= nERR_NOERROR;

(* check cycle time parameter: (CycleTime > 0) *)
IF (fCtrlCycleTime <= 0.0) THEN
	nErrorStatus := nERR_INVALIDCYCLETIME;
	bReset := TRUE;
END_IF;

(* check controller parameters: (Kp, Ki, Kd >= 0) *)
IF ((fKp < 0.0) OR (fKi < 0.0) OR (fKd < 0.0)) THEN
	nErrorStatus := nERR_INVALIDPARAM;
	bReset := TRUE;
END_IF;

(* controller reset *)
IF bReset THEN
	(* reset internal and external variables *)
	_fEOld			:= 0.0;
	fY				:= MAX(MIN(fBias, fMaxOutput), fMinOutput);
	_fYi		:= 0.0;
	_fYd		:= 0.0;
	RETURN;
END_IF

(* 3. save old variable *)
_fEOld := _fE;

(* 4. set error/deviation input *)
_fE := fSetpoint - fPresentValue;

(* 5. YP-part *)
_fYp := fKp * _fE;

(* 6. YI-part *)
_fYi := _fYi + (fKi * fCtrlCycleTime * _fE);
IF (_fYi > fMaxOutput) THEN
	(* limit wind up positive *)
	_fYi := fMaxOutput;
ELSIF (_fYi < fMinOutput) THEN
	(* limit wind up negative *)
	_fYi := fMinOutput;
END_IF

(* 7. YD-part *)
_fYd := fKd * (_fE - _fEOld) / fCtrlCycleTime;

(* 8. Ysum = YP + YI + YD + Bias and output *)
fY := _fYp + _fYi + _fYd + fBias;
fY := MAX(MIN(fY, fMaxOutput), fMinOutput);
END_FUNCTION_BLOCK

(* POU FB_BACnet_MultiStateInput, ST *)
FUNCTION_BLOCK FB_BACnet_MultiStateInput
VAR_IN_OUT
	Device	: FB_BACnet_Device;
END_VAR
VAR_OUTPUT
	bReady					: BOOL;
	nPresentValue			: UDINT;
	bOverridden				: BOOL;
	bOutOfService			: BOOL;
	bFault					: BOOL;
	bInAlarm				: BOOL;
	bError			: BOOL;
	nErrorId		: UINT;
END_VAR
VAR
	_PresentValue AT%I*: UDINT; 	(* ~(BACnet_PresentValue 	:		: )
								   		(BACnet_ObjectType 		: MI	: )	*)
	_StatusFlags AT%I*: WORD; 		(* ~(BACnet_StatusFlags 	:		: )	*)
	_StatusFlagsBits : ST_BACnet_StatusFlags;

	_nUpdateCount : UDINT := 0;
END_VAR
VAR CONSTANT
	nERR_NO_ERROR		: UINT := 0;
	nERR_WRONG_MAPPING	: UINT := 2;
	nERR_OPERATIONAL	: UINT := 3;
END_VAR
(* update server device *)
IF Device._nUpdateCount = _nUpdateCount THEN
	Device();
END_IF
(* remind current number of update counter *)
_nUpdateCount := Device._nUpdateCount;

(* check BitString format of StatusFlags --> if StatusFlags are less than 4, object isn't linked correctly *)
IF (_StatusFlags < 4) THEN
	(* wrong mapping *)
	nErrorId := nERR_WRONG_MAPPING;
	bReady := FALSE;

ELSIF Device.bOperational THEN
	(* ready state *)
	bReady := TRUE;
	nErrorId := nERR_NO_ERROR;

	(* present value *)
	nPresentValue := _PresentValue;

	(* build bit states *)
	_StatusFlagsBits := F_BACnet_StatusFlags(_StatusFlags);

	(* copy states to output *)
	bOverridden := _StatusFlagsBits.overridden;
	bOutOfService := _StatusFlagsBits.out_of_service;
	bFault := _StatusFlagsBits.fault;
	bInAlarm := _StatusFlagsBits.in_alarm;

ELSE
	(* server device not ready, reset local ready also *)
	bReady := FALSE;
	nErrorId := nERR_OPERATIONAL;
END_IF
(* set error flag *)
bError := (nErrorId <> nERR_NO_ERROR);
END_FUNCTION_BLOCK

(* POU FB_BACnet_MultiStateInput_EX, ST *)
FUNCTION_BLOCK FB_BACnet_MultiStateInput_EX
VAR_IN_OUT
	Device	: FB_BACnet_Device;
END_VAR
VAR_OUTPUT
	bReady			: BOOL;
	nPresentValue	: UDINT;
	bOverridden		: BOOL;
	bOutOfService	: BOOL;
	bFault			: BOOL;
	bInAlarm		: BOOL;
	bOverRange		: BOOL;
	bUnderRange		: BOOL;
	bNoSensor		: BOOL;
	bOpenLoop		: BOOL;
	bShortedLoop	: BOOL;
	bMultiStateFault: BOOL;
	bOtherFault		: BOOL;
	eEventState		: E_BACNETEVENTSTATE;
	bAckedTrans_ToOffNormal : BOOL;
	bAckedTrans_ToFault		: BOOL;
	bAckedTrans_ToNormal	: BOOL;
	nNbrOfStates	: UDINT;
	bError			: BOOL;
	nErrorId		: UINT;
END_VAR
VAR
	_PresentValue AT%I*: UDINT; 	(* ~(BACnet_PresentValue 	:		: )
								   		(BACnet_ObjectType 		: MI	: )	*)
	_StatusFlags AT%I*: WORD; 		(* ~(BACnet_StatusFlags 	:		: )	*)
	_StatusFlagsBits : ST_BACnet_StatusFlags;
	_EventState AT%I*: WORD; 		(* ~(BACnet_EventState 		:		: )	*)
	_Reliability AT%I*: WORD; 		(* ~(BACnet_Reliability 	:		: )	*)
	_NumberOfStates AT%I*: UDINT;	(* ~(BACnet_NumberOfStates	:		: )	*)
	_AckedTransitions AT%I*:WORD;	(* ~(BACnet_AckedTransitions:		: ) *)
	_AckedTransBits : ST_BACnet_EventTransitionBits;
	_nUpdateCount : UDINT := 0;
END_VAR
VAR CONSTANT
	nERR_NO_ERROR		: UINT := 0;
	nERR_WRONG_MAPPING	: UINT := 2;
	nERR_OPERATIONAL	: UINT := 3;
END_VAR
(* update server device *)
IF Device._nUpdateCount = _nUpdateCount THEN
	Device();
END_IF
(* remind current number of update counter *)
_nUpdateCount := Device._nUpdateCount;

(* check BitString format of StatusFlags --> if StatusFlags are less than 4, object isn't linked correctly *)
IF (_StatusFlags < 4) OR _AckedTransitions < 5 THEN
	(* wrong mapping *)
	nErrorId := nERR_WRONG_MAPPING;
	bReady := FALSE;

ELSIF Device.bOperational THEN
	(* ready state *)
	bReady := TRUE;
	nErrorId := nERR_NO_ERROR;

	(* present value *)
	nPresentValue := _PresentValue;

	(* build bit states *)
	_StatusFlagsBits := F_BACnet_StatusFlags(_StatusFlags);
	_AckedTransBits		:= F_BACnet_EventTransitionFlags(_AckedTransitions);

	(* copy states to output *)
	bOverridden := _StatusFlagsBits.overridden;
	bOutOfService := _StatusFlagsBits.out_of_service;
	bFault := _StatusFlagsBits.fault;
	bInAlarm := _StatusFlagsBits.in_alarm;
	bOverRange := (_Reliability = BACnetReliability_over_range);
	bUnderRange := (_Reliability = BACnetReliability_under_range);
	bNoSensor := (_Reliability = BACnetReliability_no_sensor);
	bOpenLoop := (_Reliability = BACnetReliability_open_loop);
	bShortedLoop := (_Reliability = BACnetReliability_shorted_loop);
	bMultiStateFault := (_Reliability = BACnetReliability_multi_state_fault);
	bOtherFault := (_Reliability = BACnetReliability_unreliable_other);
	bAckedTrans_ToOffNormal := _AckedTransBits.to_offnormal;
	bAckedTrans_ToFault := _AckedTransBits.to_fault;
	bAckedTrans_ToNormal := _AckedTransBits.to_normal;

	(* convert enumeration *)
	eEventState := _EventState;

	(* number of states *)
	nNbrOfStates := _NumberOfStates;

ELSE
	(* server device not ready, reset local ready also *)
	bReady := FALSE;
	nErrorId := nERR_OPERATIONAL;
END_IF
(* set error flag *)
bError := (nErrorId <> nERR_NO_ERROR);
END_FUNCTION_BLOCK

(* POU FB_BACnet_MultiStateOutput, ST *)
FUNCTION_BLOCK FB_BACnet_MultiStateOutput
VAR_INPUT
	bEnablePV	: BOOL; (* enable present value with priority x in priority array, FALSE = priority x disable *)
	nPV			: UDINT; (* number for priority x, when input bEnablePV is TRUE *)
END_VAR
VAR_IN_OUT
	Device	: FB_BACnet_Device;
END_VAR
VAR_OUTPUT
	bReady			: BOOL;
	nPresentValue	: UDINT;
	bOverridden		: BOOL;
	bOutOfService	: BOOL;
	bFault			: BOOL;
	bInAlarm		: BOOL;
	nNbrOfStates	: UDINT;
	bError			: BOOL;
	nErrorId		: UINT;
END_VAR
VAR
	_PresentValue AT%I*: UDINT; 			(* ~(BACnet_PresentValue 		:		: )
								   				(BACnet_ObjectType			: MO	: )	*)
	_StatusFlags AT%I*: WORD; 				(* ~(BACnet_StatusFlags			:		: )	*)
	_StatusFlagsBits : ST_BACnet_StatusFlags;
    _PresentValue_Priority12 AT%Q*: UDINT;	(* ~(BACnet_PresentValue_Priority12		:		: )	*)
	_NumberOfStates AT%I*: UDINT;			(* ~(BACnet_NumberOfStates		:		: )	*)

	_nUpdateCount : UDINT := 0;
END_VAR
VAR CONSTANT
	nERR_NO_ERROR		: UINT := 0;
	nERR_WRONG_MAPPING	: UINT := 2;
	nERR_OPERATIONAL	: UINT := 3;
END_VAR
(* update server device *)
IF Device._nUpdateCount = _nUpdateCount THEN
	Device();
END_IF
(* remind current number of update counter *)
_nUpdateCount := Device._nUpdateCount;

(* check BitString format of StatusFlags --> if StatusFlags are less than 4, object isn't linked correctly *)
IF (_StatusFlags < 4) THEN
	(* wrong mapping *)
	nErrorId := nERR_WRONG_MAPPING;
	bReady := FALSE;

ELSIF Device.bOperational THEN
	(* ready state *)
	bReady := TRUE;
	nErrorId := nERR_NO_ERROR;

	(* write into priority array *)
	IF bEnablePV THEN
		_PresentValue_Priority12	:= nPV;
	ELSE
		_PresentValue_Priority12	:= 0;
	END_IF

	(* present value *)
	nPresentValue := _PresentValue;

	(* build bit states *)
	_StatusFlagsBits := F_BACnet_StatusFlags(_StatusFlags);

	(* copy states to output *)
	bOverridden := _StatusFlagsBits.overridden;
	bOutOfService := _StatusFlagsBits.out_of_service;
	bFault := _StatusFlagsBits.fault;
	bInAlarm := _StatusFlagsBits.in_alarm;

	(* number of states *)
	nNbrOfStates := _NumberOfStates;

ELSIF Device.bFirstCycle THEN
	(* first call of the server device since reboot/reset *)
	bReady := FALSE;
	_PresentValue_Priority12 := 0;
ELSE
	(* server device not ready, reset local ready also *)
	bReady := FALSE;
	nErrorId := nERR_OPERATIONAL;
END_IF
(* set error flag *)
bError := (nErrorId <> nERR_NO_ERROR);
END_FUNCTION_BLOCK

(* POU FB_BACnet_MultiStateOutput_ADS, ST *)
FUNCTION_BLOCK FB_BACnet_MultiStateOutput_ADS
VAR_INPUT
	bEnablePV		: BOOL;
	nPV				: UDINT; (* number for priority x, when input bEnablePV is TRUE *)
	bManual			: BOOL; (* FALSE --> TRUE: write present_value immediately, FALSE: only write present_value on-change, TRUE: write present_value on-change and when device turns operational *)
	ePriority		: E_BACNETPRIORITY := BACNETPRIORITY_12;
END_VAR
VAR_IN_OUT
	Device			: FB_BACnet_Device;
END_VAR
VAR_OUTPUT
	bReady			: BOOL;
	bPvDone			: BOOL; (* present_value written over ADS *)
	nPresentValue	: UDINT;
	bOverridden		: BOOL;
	bOutOfService	: BOOL;
	bFault			: BOOL;
	bInAlarm		: BOOL;
	nNbrOfStates	: UDINT;
	bError			: BOOL;
	nErrorId		: UINT;
	nAdsErrorId		: UDINT;
END_VAR
VAR
	_PresentValue AT%I*: UDINT; 			(* ~(BACnet_PresentValue 		:		: )
								   				(BACnet_ObjectType			: MO	: )	*)
	_StatusFlags AT%I*: WORD; 				(* ~(BACnet_StatusFlags			:		: )	*)
	_StatusFlagsBits : ST_BACnet_StatusFlags;
    _PresentValue_Ads : UDINT;
	_NumberOfStates AT%I*: UDINT;			(* ~(BACnet_NumberOfStates		:		: )	*)
	_ObjectId AT%I*: DWORD;					(* ~(BACnet_ObjectIdentifier			 :		: LINK) *)
	_nUpdateCount : UDINT := 0;
	_WriteProp : FB_BACnet_WriteProp;
	_rtrigManual : R_TRIG;
	_bEnPvOld : BOOL;
	_nObjType : E_BACNETOBJECTTYPE;
END_VAR
VAR CONSTANT
	nERR_NO_ERROR		: UINT := 0;
	nERR_WRONG_MAPPING	: UINT := 2;
	nERR_OPERATIONAL	: UINT := 3;
	nERR_WRONG_TYPE		: UINT := 4;
END_VAR
(* update server device *)
IF Device._nUpdateCount = _nUpdateCount THEN
	Device();
END_IF
(* remind current number of update counter *)
_nUpdateCount := Device._nUpdateCount;

(* trigger on manual flag *)
_rtrigManual(CLK:= bManual, Q=> );

(* decode object type *)
_nObjType := F_BACnet_GetObjType(_ObjectId);

(* check BitString format of StatusFlags --> if StatusFlags are less than 4, object isn't linked correctly *)
IF _nObjType <> BACnetObjectType_MultiStateOutput THEN
	(* wrong mapped object type *)
	nErrorId := nERR_WRONG_TYPE;
	bReady := FALSE;
	bPvDone := FALSE;

ELSIF (_StatusFlags < 4) THEN
	(* wrong mapping *)
	nErrorId := nERR_WRONG_MAPPING;
	bReady := FALSE;
	bPvDone := FALSE;

ELSIF Device.bOperational THEN
	(* write present_value on manual trigger, on-change and on operational recover *)
	IF		_rtrigManual.Q
		OR	((F_BACnet_IsFinite(_PresentValue_Ads) <> F_BACnet_IsFinite(_PresentValue_Ads)) AND bEnablePV)
		OR	((nPV <> _PresentValue_Ads) AND bEnablePV)
		OR	((NOT bReady) AND bManual)
		OR	(bEnablePV <> _bEnPvOld)
	THEN
		_WriteProp.bExecute := TRUE;
		bPvDone := FALSE;
		(* write depending on enable state *)
		IF bEnablePV THEN
			_PresentValue_Ads := nPV;
		ELSE
			_PresentValue_Ads := 0;
		END_IF
		_bEnPvOld := bEnablePV;
	END_IF

	(* ready state *)
	bReady := TRUE;
	nErrorId := nERR_NO_ERROR;

	(* present value *)
	nPresentValue := _PresentValue;

	(* build bit states *)
	_StatusFlagsBits := F_BACnet_StatusFlags(_StatusFlags);

	(* copy states to output *)
	bOverridden := _StatusFlagsBits.overridden;
	bOutOfService := _StatusFlagsBits.out_of_service;
	bFault := _StatusFlagsBits.fault;
	bInAlarm := _StatusFlagsBits.in_alarm;

	(* number of states *)
	nNbrOfStates := _NumberOfStates;

ELSIF Device.bFirstCycle THEN
	(* first call of the server device since reboot/reset *)
	bReady := FALSE;
	bPvDone := FALSE;
ELSE
	(* server device not ready, reset local ready also *)
	bReady := FALSE;
	nErrorId := nERR_OPERATIONAL;
	bPvDone := FALSE;
END_IF

(* call write property command *)
_WriteProp(
	BACnetDevicePort	:= Device.nAdsPort,
	bExecute			:= ,
	sNetId				:= Device.sAmsNetId,
	ObjectType			:= _nObjType,
	PropertyID			:= BACnetPropertyIdentifier_PresentValue,
	Priority			:= ePriority,
	DataType			:= BACnetDataType_UnsignedInteger,
	ObjectInstance		:= F_BACnet_GetObjInstance(_ObjectId),
	ptrValue			:= ADR(_PresentValue_Ads),
	nLenValue			:= SIZEOF(_PresentValue_Ads),
	bDone				=> ,
	bBusy				=> ,
	bError				=> ,
	nErrID				=> nAdsErrorId);

(* set done flag *)
IF _WriteProp.bExecute AND (NOT _WriteProp.bBusy) THEN
	(* reset execution bit *)
	_WriteProp(bExecute := FALSE);
	(* check if command was finished with error *)
	IF _WriteProp.bError THEN
		IF bManual THEN
			(* retrigger if manual flag is set *)
			_WriteProp.bExecute := TRUE;
		END_IF
		bPvDone := FALSE;
	ELSE
		(* successful written *)
		bPvDone	:= TRUE;
	END_IF
END_IF

(* set error flag *)
bError := (nErrorId <> nERR_NO_ERROR) OR (nAdsErrorId <> 0);
END_FUNCTION_BLOCK

(* POU FB_BACnet_MultiStateOutput_EX, ST *)
FUNCTION_BLOCK FB_BACnet_MultiStateOutput_EX
VAR_INPUT
	bEnablePV		: BOOL; (* enable present value with priority x in priority array, FALSE = priority x disable *)
	nPV		: UDINT; (* number for priority x, when input bEnablePV is TRUE *)
END_VAR
VAR_IN_OUT
	Device	: FB_BACnet_Device;
END_VAR
VAR_OUTPUT
	bReady			: BOOL;
	nPresentValue	: UDINT;
	bOverridden		: BOOL;
	bOutOfService	: BOOL;
	bFault			: BOOL;
	bInAlarm		: BOOL;
	bNoOutput		: BOOL;
	bOpenLoop		: BOOL;
	bShortedLoop	: BOOL;
	bOtherFault		: BOOL;
	eEventState		: E_BACNETEVENTSTATE;
	bAckedTrans_ToOffNormal : BOOL;
	bAckedTrans_ToFault		: BOOL;
	bAckedTrans_ToNormal	: BOOL;
	nActivePrio		: UINT;
	nNbrOfStates	: UDINT;
	bError			: BOOL;
	nErrorId		: UINT;
END_VAR
VAR
	_PresentValue AT%I*: UDINT; 			(* ~(BACnet_PresentValue 		:		: )
								   				(BACnet_ObjectType			: MO	: )	*)
	_StatusFlags AT%I*: WORD; 				(* ~(BACnet_StatusFlags			:		: )	*)
	_StatusFlagsBits : ST_BACnet_StatusFlags;
	_EventState AT%I*: WORD;				(* ~(BACnet_EventState			:		: )	*)
	_Reliability AT%I*: WORD; 				(* ~(BACnet_Reliability			:		: )	*)
    _PresentValue_Priority12 AT%Q*: UDINT;	(* ~(BACnet_PresentValue_Priority12		:		: )	*)
	_ActivePriority AT%I*: UDINT; 			(* ~(BACnet_ActivePriority 		:		: )	*)
	_NumberOfStates AT%I*: UDINT;			(* ~(BACnet_NumberOfStates		:		: )	*)
	_AckedTransitions AT%I*:WORD;			(* ~(BACnet_AckedTransitions:		: ) *)
	_AckedTransBits : ST_BACnet_EventTransitionBits;
	_nUpdateCount : UDINT := 0;
END_VAR
VAR CONSTANT
	nERR_NO_ERROR		: UINT := 0;
	nERR_WRONG_MAPPING	: UINT := 2;
	nERR_OPERATIONAL	: UINT := 3;
END_VAR
(* update server device *)
IF Device._nUpdateCount = _nUpdateCount THEN
	Device();
END_IF
(* remind current number of update counter *)
_nUpdateCount := Device._nUpdateCount;

(* check BitString format of StatusFlags --> if StatusFlags are less than 4, object isn't linked correctly *)
IF (_StatusFlags < 4) OR _AckedTransitions < 5 THEN
	(* wrong mapping *)
	nErrorId := nERR_WRONG_MAPPING;
	bReady := FALSE;

ELSIF Device.bOperational THEN
	(* ready state *)
	bReady := TRUE;
	nErrorId := nERR_NO_ERROR;

	(* write into priority array *)
	IF bEnablePV THEN
		_PresentValue_Priority12	:= nPV;
	ELSE
		_PresentValue_Priority12	:= 0;
	END_IF

	(* present value *)
	nPresentValue := _PresentValue;

	(* build bit states *)
	_StatusFlagsBits := F_BACnet_StatusFlags(_StatusFlags);
	_AckedTransBits		:= F_BACnet_EventTransitionFlags(_AckedTransitions);

	(* copy states to output *)
	bOverridden := _StatusFlagsBits.overridden;
	bOutOfService := _StatusFlagsBits.out_of_service;
	bFault := _StatusFlagsBits.fault;
	bInAlarm := _StatusFlagsBits.in_alarm;
	bNoOutput := (_Reliability = BACnetReliability_no_output);
	bOpenLoop := (_Reliability = BACnetReliability_open_loop);
	bShortedLoop := (_Reliability = BACnetReliability_shorted_loop);
	bOtherFault := (_Reliability = BACnetReliability_unreliable_other);
	bAckedTrans_ToOffNormal := _AckedTransBits.to_offnormal;
	bAckedTrans_ToFault := _AckedTransBits.to_fault;
	bAckedTrans_ToNormal := _AckedTransBits.to_normal;

	(* convert enumeration *)
	eEventState := _EventState;

	(* copy active priority *)
	nActivePrio := UDINT_TO_UINT(_ActivePriority);

	(* number of states *)
	nNbrOfStates := _NumberOfStates;

ELSIF Device.bFirstCycle THEN
	(* first call of the server device since reboot/reset *)
	bReady := FALSE;
	_PresentValue_Priority12 := 0;
ELSE
	(* server device not ready, reset local ready also *)
	bReady := FALSE;
	nErrorId := nERR_OPERATIONAL;
END_IF
(* set error flag *)
bError := (nErrorId <> nERR_NO_ERROR);
END_FUNCTION_BLOCK

(* POU FB_BACnet_MultiStateValue, ST *)
FUNCTION_BLOCK FB_BACnet_MultiStateValue
VAR_INPUT
	bEnablePV	: BOOL; (* enable present value with priority x in priority array, FALSE = priority x disable *)
	nPV			: UDINT; (* number for priority x, when input bEnablePV is TRUE *)
END_VAR
VAR_IN_OUT
	Device	: FB_BACnet_Device;
END_VAR
VAR_OUTPUT
	bReady			: BOOL;
	nPresentValue	: UDINT;
	bOverridden		: BOOL;
	bOutOfService	: BOOL;
	bFault			: BOOL;
	bInAlarm		: BOOL;
	nNbrOfStates	: UDINT;
	bError			: BOOL;
	nErrorId		: UINT;
END_VAR
VAR
	_PresentValue AT%I*: UDINT; 			(* ~(BACnet_PresentValue 	:		: )
								   				(BACnet_ObjectType 		: MV	: )	*)
	_StatusFlags AT%I*: WORD; 				(* ~(BACnet_StatusFlags 	:		: )	*)
	_StatusFlagsBits : ST_BACnet_StatusFlags;
    _PresentValue_Priority12 AT%Q*: UDINT;	(* ~(BACnet_PresentValue_Priority12	:		: )	*)
	_NumberOfStates AT%I*: UDINT;			(* ~(BACnet_NumberOfStates	:		: )	*)
	_nUpdateCount : UDINT := 0;
END_VAR
VAR CONSTANT
	nERR_NO_ERROR		: UINT := 0;
	nERR_WRONG_MAPPING	: UINT := 2;
	nERR_OPERATIONAL	: UINT := 3;
END_VAR
(* update server device *)
IF Device._nUpdateCount = _nUpdateCount THEN
	Device();
END_IF
(* remind current number of update counter *)
_nUpdateCount := Device._nUpdateCount;

(* check BitString format of StatusFlags --> if StatusFlags are less than 4, object isn't linked correctly *)
IF (_StatusFlags < 4) THEN
	(* wrong mapping *)
	nErrorId := nERR_WRONG_MAPPING;
	bReady := FALSE;

ELSIF Device.bOperational THEN
	(* ready state *)
	bReady := TRUE;
	nErrorId := nERR_NO_ERROR;

	(* write into priority array *)
	IF bEnablePV THEN
		_PresentValue_Priority12	:= nPV;
	ELSE
		_PresentValue_Priority12	:= 0;
	END_IF

	(* present value *)
	nPresentValue := _PresentValue;

	(* build bit states *)
	_StatusFlagsBits := F_BACnet_StatusFlags(_StatusFlags);

	(* copy states to output *)
	bOverridden := _StatusFlagsBits.overridden;
	bOutOfService := _StatusFlagsBits.out_of_service;
	bFault := _StatusFlagsBits.fault;
	bInAlarm := _StatusFlagsBits.in_alarm;

	(* number of states *)
	nNbrOfStates := _NumberOfStates;

ELSIF Device.bFirstCycle THEN
	(* first call of the server device since reboot/reset *)
	bReady := FALSE;
	_PresentValue_Priority12 := 0;
ELSE
	(* server device not ready, reset local ready also *)
	bReady := FALSE;
	nErrorId := nERR_OPERATIONAL;
END_IF
(* set error flag *)
bError := (nErrorId <> nERR_NO_ERROR);
END_FUNCTION_BLOCK

(* POU FB_BACnet_MultiStateValue_ADS, ST *)
FUNCTION_BLOCK FB_BACnet_MultiStateValue_ADS
VAR_INPUT
	bEnablePV		: BOOL;
	nPV				: UDINT; (* number for priority x, when input bEnablePV is TRUE *)
	bManual			: BOOL; (* FALSE --> TRUE: write present_value immediately, FALSE: only write present_value on-change, TRUE: write present_value on-change and when device turns operational *)
	ePriority		: E_BACNETPRIORITY := BACNETPRIORITY_12;
END_VAR
VAR_IN_OUT
	Device			: FB_BACnet_Device;
END_VAR
VAR_OUTPUT
	bReady			: BOOL;
	bPvDone			: BOOL; (* present_value written over ADS *)
	nPresentValue	: UDINT;
	bOverridden		: BOOL;
	bOutOfService	: BOOL;
	bFault			: BOOL;
	bInAlarm		: BOOL;
	nNbrOfStates	: UDINT;
	bError			: BOOL;
	nErrorId		: UINT;
	nAdsErrorId		: UDINT;
END_VAR
VAR
	_PresentValue AT%I*: UDINT; 			(* ~(BACnet_PresentValue 	:		: )
								   				(BACnet_ObjectType 		: MV	: )	*)
	_StatusFlags AT%I*: WORD; 				(* ~(BACnet_StatusFlags 	:		: )	*)
	_StatusFlagsBits : ST_BACnet_StatusFlags;
    _PresentValue_Ads : UDINT;
	_NumberOfStates AT%I*: UDINT;			(* ~(BACnet_NumberOfStates	:		: )	*)
	_ObjectId AT%I*: DWORD;					(* ~(BACnet_ObjectIdentifier			 :		: LINK) *)
	_nUpdateCount : UDINT := 0;
	_WriteProp : FB_BACnet_WriteProp;
	_rtrigManual : R_TRIG;
	_bEnPvOld : BOOL;
	_nObjType : E_BACNETOBJECTTYPE;
END_VAR
VAR CONSTANT
	nERR_NO_ERROR		: UINT := 0;
	nERR_WRONG_MAPPING	: UINT := 2;
	nERR_OPERATIONAL	: UINT := 3;
	nERR_WRONG_TYPE		: UINT := 4;
END_VAR
(* update server device *)
IF Device._nUpdateCount = _nUpdateCount THEN
	Device();
END_IF
(* remind current number of update counter *)
_nUpdateCount := Device._nUpdateCount;

(* trigger on manual flag *)
_rtrigManual(CLK:= bManual, Q=> );

(* decode object type *)
_nObjType := F_BACnet_GetObjType(_ObjectId);

(* check BitString format of StatusFlags --> if StatusFlags are less than 4, object isn't linked correctly *)
IF _nObjType <> BACnetObjectType_MultiStateValue THEN
	(* wrong mapped object type *)
	nErrorId := nERR_WRONG_TYPE;
	bReady := FALSE;
	bPvDone := FALSE;

ELSIF (_StatusFlags < 4) THEN
	(* wrong mapping *)
	nErrorId := nERR_WRONG_MAPPING;
	bReady := FALSE;
	bPvDone := FALSE;

ELSIF Device.bOperational THEN
	(* write present_value on manual trigger, on-change and on operational recover *)
	IF		_rtrigManual.Q
		OR	((F_BACnet_IsFinite(_PresentValue_Ads) <> F_BACnet_IsFinite(_PresentValue_Ads)) AND bEnablePV)
		OR	((nPV <> _PresentValue_Ads) AND bEnablePV)
		OR	((NOT bReady) AND bManual)
		OR	(bEnablePV <> _bEnPvOld)
	THEN
		_WriteProp.bExecute := TRUE;
		bPvDone := FALSE;
		(* write depending on enable state *)
		IF bEnablePV THEN
			_PresentValue_Ads := nPV;
		ELSE
			_PresentValue_Ads := 0;
		END_IF
		_bEnPvOld := bEnablePV;
	END_IF

	(* ready state *)
	bReady := TRUE;
	nErrorId := nERR_NO_ERROR;

	(* present value *)
	nPresentValue := _PresentValue;

	(* build bit states *)
	_StatusFlagsBits := F_BACnet_StatusFlags(_StatusFlags);

	(* copy states to output *)
	bOverridden := _StatusFlagsBits.overridden;
	bOutOfService := _StatusFlagsBits.out_of_service;
	bFault := _StatusFlagsBits.fault;
	bInAlarm := _StatusFlagsBits.in_alarm;

	(* number of states *)
	nNbrOfStates := _NumberOfStates;

ELSIF Device.bFirstCycle THEN
	(* first call of the server device since reboot/reset *)
	bReady := FALSE;
	bPvDone := FALSE;
ELSE
	(* server device not ready, reset local ready also *)
	bReady := FALSE;
	nErrorId := nERR_OPERATIONAL;
	bPvDone := FALSE;
END_IF

(* call write property command *)
_WriteProp(
	BACnetDevicePort	:= Device.nAdsPort,
	bExecute			:= ,
	sNetId				:= Device.sAmsNetId,
	ObjectType			:= _nObjType,
	PropertyID			:= BACnetPropertyIdentifier_PresentValue,
	Priority			:= ePriority,
	DataType			:= BACnetDataType_UnsignedInteger,
	ObjectInstance		:= F_BACnet_GetObjInstance(_ObjectId),
	ptrValue			:= ADR(_PresentValue_Ads),
	nLenValue			:= SIZEOF(_PresentValue_Ads),
	bDone				=> ,
	bBusy				=> ,
	bError				=> ,
	nErrID				=> nAdsErrorId);

(* set done flag *)
IF _WriteProp.bExecute AND (NOT _WriteProp.bBusy) THEN
	(* reset execution bit *)
	_WriteProp(bExecute := FALSE);
	(* check if command was finished with error *)
	IF _WriteProp.bError THEN
		IF bManual THEN
			(* retrigger if manual flag is set *)
			_WriteProp.bExecute := TRUE;
		END_IF
		bPvDone := FALSE;
	ELSE
		(* successful written *)
		bPvDone	:= TRUE;
	END_IF
END_IF

(* set error flag *)
bError := (nErrorId <> nERR_NO_ERROR) OR (nAdsErrorId <> 0);
END_FUNCTION_BLOCK

(* POU FB_BACnet_MultiStateValue_EX, ST *)
FUNCTION_BLOCK FB_BACnet_MultiStateValue_EX
VAR_INPUT
	bEnablePV	: BOOL; (* enable present value with priority x in priority array, FALSE = priority x disable *)
	nPV			: UDINT; (* number for priority x, when input bEnablePV is TRUE *)
END_VAR
VAR_IN_OUT
	Device		: FB_BACnet_Device;
END_VAR
VAR_OUTPUT
	bReady			: BOOL;
	nPresentValue	: UDINT;
	bOverridden		: BOOL;
	bOutOfService	: BOOL;
	bFault			: BOOL;
	bInAlarm		: BOOL;
	bMultiStateFault: BOOL;
	bOtherFault		: BOOL;
	eEventState		: E_BACNETEVENTSTATE;
	bAckedTrans_ToOffNormal : BOOL;
	bAckedTrans_ToFault		: BOOL;
	bAckedTrans_ToNormal	: BOOL;
	nActivePrio		: UINT;
	nNbrOfStates	: UDINT;
	bError			: BOOL;
	nErrorId		: UINT;
END_VAR
VAR
	_PresentValue AT%I*: UDINT; 			(* ~(BACnet_PresentValue 	:		: )
								   				(BACnet_ObjectType 		: MV	: )	*)
	_StatusFlags AT%I*: WORD; 				(* ~(BACnet_StatusFlags 	:		: )	*)
	_StatusFlagsBits : ST_BACnet_StatusFlags;
	_EventState AT%I*: WORD;				(* ~(BACnet_EventState 		:		: )	*)
	_Reliability AT%I*: WORD;				(* ~(BACnet_Reliability 	:		: )	*)
    _PresentValue_Priority12 AT%Q*: UDINT;	(* ~(BACnet_PresentValue_Priority12	:		: )	*)
	_ActivePriority AT%I*: UDINT; 			(* ~(BACnet_ActivePriority 	:		: )	*)
	_NumberOfStates AT%I*: UDINT;			(* ~(BACnet_NumberOfStates	:		: )	*)
	_AckedTransitions AT%I*:WORD;			(* ~(BACnet_AckedTransitions:		: ) *)
	_AckedTransBits : ST_BACnet_EventTransitionBits;
	_nUpdateCount : UDINT := 0;
END_VAR
VAR CONSTANT
	nERR_NO_ERROR		: UINT := 0;
	nERR_WRONG_MAPPING	: UINT := 2;
	nERR_OPERATIONAL	: UINT := 3;
END_VAR
(* update server device *)
IF Device._nUpdateCount = _nUpdateCount THEN
	Device();
END_IF
(* remind current number of update counter *)
_nUpdateCount := Device._nUpdateCount;

(* check BitString format of StatusFlags --> if StatusFlags are less than 4, object isn't linked correctly *)
IF (_StatusFlags < 4) OR _AckedTransitions < 5 THEN
	(* wrong mapping *)
	nErrorId := nERR_WRONG_MAPPING;
	bReady := FALSE;

ELSIF Device.bOperational THEN
	(* ready state *)
	bReady := TRUE;
	nErrorId := nERR_NO_ERROR;

	(* write into priority array *)
	IF bEnablePV THEN
		_PresentValue_Priority12	:= nPV;
	ELSE
		_PresentValue_Priority12	:= 0;
	END_IF

	(* present value *)
	nPresentValue := _PresentValue;

	(* build bit states *)
	_StatusFlagsBits := F_BACnet_StatusFlags(_StatusFlags);
	_AckedTransBits		:= F_BACnet_EventTransitionFlags(_AckedTransitions);

	(* copy states to output *)
	bOverridden := _StatusFlagsBits.overridden;
	bOutOfService := _StatusFlagsBits.out_of_service;
	bFault := _StatusFlagsBits.fault;
	bInAlarm := _StatusFlagsBits.in_alarm;
	bMultiStateFault := (_Reliability = BACnetReliability_multi_state_fault);
	bOtherFault := (_Reliability = BACnetReliability_unreliable_other);
	bAckedTrans_ToOffNormal := _AckedTransBits.to_offnormal;
	bAckedTrans_ToFault := _AckedTransBits.to_fault;
	bAckedTrans_ToNormal := _AckedTransBits.to_normal;

	(* convert enumeration *)
	eEventState := _EventState;

	(* copy active priority *)
	nActivePrio := UDINT_TO_UINT(_ActivePriority);

	(* number of states *)
	nNbrOfStates := _NumberOfStates;

ELSIF Device.bFirstCycle THEN
	(* first call of the server device since reboot/reset *)
	bReady := FALSE;
	_PresentValue_Priority12 := 0;
ELSE
	(* server device not ready, reset local ready also *)
	bReady := FALSE;
	nErrorId := nERR_OPERATIONAL;
END_IF
(* set error flag *)
bError := (nErrorId <> nERR_NO_ERROR);
END_FUNCTION_BLOCK

(* POU FB_BACnet_NotificationClass, ST *)
FUNCTION_BLOCK FB_BACnet_NotificationClass
VAR_IN_OUT
	Device	: FB_BACnet_Device;
END_VAR
VAR_OUTPUT
	bReady			: BOOL;
	bError			: BOOL;
	nErrorId		: UINT;
END_VAR
VAR
	_ObjectType		: E_BACNETOBJECTTYPE; (* ~(BACNET_OBJECTTYPE :NC:)  *)
	_nUpdateCount	: UDINT := 0;
END_VAR
VAR CONSTANT
	nERR_NO_ERROR		: UINT := 0;
	nERR_OPERATIONAL	: UINT := 3;
END_VAR
_ObjectType := BACnetObjectType_NotificationClass;
(* update server device *)
IF Device._nUpdateCount = _nUpdateCount THEN
	Device();
END_IF
(* remind current number of update counter *)
_nUpdateCount := Device._nUpdateCount;

IF Device.bOperational THEN
	(* ready state *)
	bReady := TRUE;
	nErrorId := nERR_NO_ERROR;
ELSE
	(* server device not ready, reset local ready also *)
	bReady := FALSE;
	nErrorId := nERR_OPERATIONAL;
END_IF
(* set error flag *)
bError := (nErrorId <> nERR_NO_ERROR);
END_FUNCTION_BLOCK

(* POU FB_BACnet_NotificationSinkDelEntry, ST *)
FUNCTION_BLOCK FB_BACnet_NotificationSinkDelEntry
VAR_INPUT
	bExecute	: BOOL;
	nIndex		: UDINT;
	sNetId		: T_AmsNetId;
	nPort		: T_AmsPort;
	tTimeout	: TIME := tBACnet_ADSTimeOut;
END_VAR
VAR_OUTPUT
	bBusy		: BOOL;
	bEmpty		: BOOL;
	bError		: BOOL;
	nErrorId	: UDINT;
END_VAR
VAR
	_AdsReadClient	: ADSREAD;
END_VAR
	_AdsReadClient(
		NETID	:= sNetId,
		PORT	:= nPort,
		IDXGRP	:= 16#5,
		IDXOFFS	:= nIndex,
		LEN		:= 0,
		DESTADDR:= 0,
		READ	:= bExecute,
		TMOUT	:= tTimeout,
		BUSY	=> bBusy,
		ERR		=> bError,
		ERRID	=> nErrorId);

	bEmpty := ((UDINT_TO_DWORD(_AdsReadClient.ERRID) AND 16#FFF) = 16#703);
END_FUNCTION_BLOCK

(* POU FB_BACnet_Program, ST *)
FUNCTION_BLOCK FB_BACnet_Program
VAR_INPUT
	bRelease			: BOOL;
	bCommonError		: BOOL;
	bWaitForSomething	: BOOL;
	stDoneFlags			: ST_BACnet_ProgramHandshakeRequests;
	stFailedFlags		: ST_BACnet_ProgramHandshakeRequests;
	bModeUnloadComplex	: BOOL := TRUE;
END_VAR
VAR_IN_OUT
	Device	: FB_BACnet_Device;
END_VAR
VAR_OUTPUT
	bReady			: BOOL;
	bOverridden		: BOOL;
	bOutOfService	: BOOL;
	bFault			: BOOL;
	bInAlarm		: BOOL;
	bProcessError	: BOOL;
	bOtherFault		: BOOL;
	stRequestFlags	: ST_BACnet_ProgramHandshakeRequests;
	stActiveStateFlags	: ST_BACnet_ProgramHandshakeStates;
	bError			: BOOL;
	nErrorId		: UINT;
END_VAR
VAR
(* from BACnet to PLC *)
	_ProgramChange AT%I*: WORD;			(* ~(BACnet_ProgramChange 				 :		: )
			   								(BACnet_ObjectType 					 : PROG	: ) *)
	_StatusFlags AT%I*: WORD;			(* ~(BACnet_StatusFlags 				 :		: )	*)
	_StatusFlagsBits 	: ST_BACnet_StatusFlags;
	_Reliability AT%I*: WORD;			(* ~(BACnet_Reliability 				 :		: )	*)

(* from PLC to BACnet *)
	_SetProgramReadyState AT%Q*: BOOL;	(* ~ (BACnet_SetProgramReadyState 		 :		: )	*)
	_ProgramState AT%Q*: WORD;			(* ~(BACnet_ProgramState 				 :		: ) *)
	_ReasonForHalt AT%Q*: WORD;			(* ~(BACnet_ReasonForHalt 				 : 		: )	*)

(* internal signals *)
	_bTriggerSetup		: BOOL;
	_ActiveChange		: E_BACNETPROGRAMREQUEST; (* ACTIVE PROGRAM CHANGE *)
	_bLockedForChange	: BOOL;
	_nUpdateCount		: UDINT := 0;
END_VAR
VAR CONSTANT
	nERR_NO_ERROR		: UINT := 0;
	nERR_WRONG_MAPPING	: UINT := 2;
	nERR_OPERATIONAL	: UINT := 3;
END_VAR
(* update server device *)
IF Device._nUpdateCount = _nUpdateCount THEN
	Device();
END_IF
(* remind current number of update counter *)
_nUpdateCount := Device._nUpdateCount;

(* check BitString format of StatusFlags --> if StatusFlags are less than 4, object isn't linked correctly *)
IF (_StatusFlags < 4) THEN
	(* wrong mapping *)
	nErrorId := nERR_WRONG_MAPPING;
	bReady := FALSE;

ELSIF Device.bOperational THEN
	(* ready state *)
	bReady := TRUE;
	nErrorId := nERR_NO_ERROR;

	(* decode status flags *)
	_StatusFlagsBits := F_BACnet_StatusFlags(_StatusFlags);

	(* copy states to output *)
	bOverridden := _StatusFlagsBits.overridden;
	bOutOfService := _StatusFlagsBits.out_of_service;
	bFault := _StatusFlagsBits.fault;
	bInAlarm := _StatusFlagsBits.in_alarm;
	bProcessError := (_Reliability = BACnetReliability_process_error);
	bOtherFault := (_Reliability = BACnetReliability_unreliable_other);

	(* execute change *)
	CASE _ActiveChange OF
		BACnetProgramRequest_ready:
			(* idle *);

		BACnetProgramRequest_load:
			_ProgramState	:= BACnetProgramState_loading;
			_ActiveChange	:= BACnetProgramRequest_ready;

		BACnetProgramRequest_restart,
		BACnetProgramRequest_run:
			IF _bTriggerSetup THEN
				(* wait on setup finish *)
				IF stFailedFlags.bSetup OR bCommonError OR (NOT bRelease) THEN
					(* abort *)
					_ProgramState := BACnetProgramState_halted;
					_ActiveChange := BACnetProgramRequest_ready;
					_ReasonForHalt := BACnetProgramError_progerror_internal;
				ELSIF stDoneFlags.bSetup THEN
					(* setup done, start "normal" running mode *)
					_bTriggerSetup := FALSE;
					_ActiveChange := BACnetProgramRequest_run;
				END_IF
			ELSE
				IF stFailedFlags.bRun OR bCommonError OR (NOT bRelease) THEN
					(* abort *)
					_ProgramState := BACnetProgramState_halted;
					_ActiveChange := BACnetProgramRequest_ready;
					_ReasonForHalt := BACnetProgramError_progerror_internal;
				ELSIF stDoneFlags.bRun THEN
					(* switch to running state *)
					_ProgramState := BACnetProgramState_running;
					_ActiveChange := BACnetProgramRequest_ready;
				END_IF
			END_IF

		BACnetProgramRequest_halt:
			(* wait on halted *)
			IF stFailedFlags.bHalt OR bCommonError OR (NOT bRelease) THEN
				(* abort *)
				_ProgramState := BACnetProgramState_halted;
				_ActiveChange := BACnetProgramRequest_ready;
				_ReasonForHalt := BACnetProgramError_progerror_internal;
			ELSIF stDoneFlags.bHalt THEN
				(* halted *)
				_ProgramState := BACnetProgramState_halted;
				_ActiveChange := BACnetProgramRequest_ready;
				_ReasonForHalt := BACnetProgramError_program;
			END_IF

		BACnetProgramRequest_unload:
			_ProgramState	:= BACnetProgramState_unloading;
			_ActiveChange	:= BACnetProgramRequest_ready;

	END_CASE

	(* start change request and handle error states *)
	IF (_ActiveChange = BACnetProgramRequest_ready) THEN

		CASE _ProgramState OF
			BACnetProgramState_idle:
				IF bCommonError THEN
					(* abort *)
					_ProgramState := BACnetProgramState_halted;
					_ReasonForHalt := BACnetProgramError_progerror_internal;
				ELSIF (NOT bRelease) THEN
					(* abort *)
					_ProgramState := BACnetProgramState_halted;
					_ReasonForHalt := BACnetProgramError_other;
				ELSIF (NOT _bLockedForChange) THEN
					_ReasonForHalt := BACnetProgramError_program_normal;
					CASE _ProgramChange OF
						BACnetProgramRequest_unload,
						BACnetProgramRequest_halt:
							(* acknowledge without execution *)
							_SetProgramReadyState	:= TRUE;
						BACnetProgramRequest_restart,
						BACnetProgramRequest_run,
						BACnetProgramRequest_load:
							(* execute request *)
							_ActiveChange := BACnetProgramRequest_load;
							_bTriggerSetup := TRUE;
					END_CASE
				END_IF

			BACnetProgramState_loading:
				IF bCommonError THEN
					(* abort *)
					_ProgramState := BACnetProgramState_halted;
					_ReasonForHalt := BACnetProgramError_progerror_internal;
				ELSIF (NOT bRelease) THEN
					(* abort *)
					_ProgramState := BACnetProgramState_halted;
					_ReasonForHalt := BACnetProgramError_other;
				ELSIF stFailedFlags.bLoad THEN
					(* abort *)
					_ProgramState := BACnetProgramState_halted;
					_ReasonForHalt := BACnetProgramError_load_failed;
				ELSIF stDoneFlags.bLoad THEN
					(* DONE *)
					_bTriggerSetup := TRUE;
					_ActiveChange := BACnetProgramRequest_run;
				ELSIF (NOT _bLockedForChange) THEN
					_ReasonForHalt := BACnetProgramError_program_normal;
					CASE _ProgramChange OF
						BACnetProgramRequest_load,
						BACnetProgramRequest_run,
						BACnetProgramRequest_halt,
						BACnetProgramRequest_restart:
							(* acknowledge without execution *)
							_SetProgramReadyState	:= TRUE;
						BACnetProgramRequest_unload:
							(* execute request *)
							_ActiveChange := _ProgramChange;
					END_CASE
				END_IF

			BACnetProgramState_running:
				IF bCommonError THEN
					(* abort *)
					_ProgramState := BACnetProgramState_halted;
					_ReasonForHalt := BACnetProgramError_progerror_internal;
				ELSIF (NOT bRelease) THEN
					(* abort *)
					_ProgramState := BACnetProgramState_halted;
					_ReasonForHalt := BACnetProgramError_other;
				ELSIF bWaitForSomething THEN
					(* wait on something *)
					_ProgramState := BACnetProgramState_waiting;
				ELSIF (NOT _bLockedForChange) THEN
					_ReasonForHalt := BACnetProgramError_program_normal;
					CASE _ProgramChange OF
						BACnetProgramRequest_run:
							(* is already running *)
							_SetProgramReadyState	:= TRUE;
						BACnetProgramRequest_unload,
						BACnetProgramRequest_halt:
							(* execute request *)
							_ActiveChange := _ProgramChange;
						BACnetProgramRequest_restart,
						BACnetProgramRequest_load:
							(* retrigger setup *)
							_ActiveChange := BACnetProgramRequest_restart;
							_bTriggerSetup := TRUE;
					END_CASE
				END_IF

			BACnetProgramState_waiting:
				IF bCommonError THEN
					(* abort *)
					_ProgramState := BACnetProgramState_halted;
					_ReasonForHalt := BACnetProgramError_progerror_internal;
				ELSIF (NOT bRelease) THEN
					(* abort *)
					_ProgramState := BACnetProgramState_halted;
					_ReasonForHalt := BACnetProgramError_other;
				ELSIF (NOT bWaitForSomething) THEN
					(* got it *)
					_ProgramState := BACnetProgramState_running;
				ELSIF (NOT _bLockedForChange) THEN
					_ReasonForHalt := BACnetProgramError_program_normal;
					CASE _ProgramChange OF
						BACnetProgramRequest_run:
							(* is already running *)
							_SetProgramReadyState	:= TRUE;
						BACnetProgramRequest_unload,
						BACnetProgramRequest_halt:
							(* execute request *)
							_ActiveChange := _ProgramChange;
					END_CASE
				END_IF

			BACnetProgramState_halted:
				IF (NOT bCommonError) AND bRelease AND (NOT _bLockedForChange) THEN
					CASE _ProgramChange OF
						BACnetProgramRequest_halt:
							(* acknowledge without execution *)
							_SetProgramReadyState	:= TRUE;
						BACnetProgramRequest_unload:
							(* execute request *)
							_ActiveChange := _ProgramChange;
						BACnetProgramRequest_restart,
						BACnetProgramRequest_load:
							(* retrigger setup *)
							_ActiveChange := BACnetProgramRequest_restart;
							_bTriggerSetup := TRUE;
						BACnetProgramRequest_run:
							(* start, but don't trigger setup *)
							_ActiveChange := _ProgramChange;
							_bTriggerSetup := FALSE;
					END_CASE
				END_IF

			BACnetProgramState_unloading:
				IF bModeUnloadComplex THEN
					_ReasonForHalt := BACnetProgramError_program_normal;
					IF bCommonError THEN
						(* abort *)
						_ProgramState := BACnetProgramState_halted;
						_ActiveChange := BACnetProgramRequest_ready;
						_ReasonForHalt := BACnetProgramError_progerror_internal;
					ELSIF (NOT bRelease) THEN
						(* abort *)
						_ProgramState := BACnetProgramState_halted;
						_ActiveChange := BACnetProgramRequest_ready;
						_ReasonForHalt := BACnetProgramError_other;
					ELSIF stFailedFlags.bUnload THEN
						(* abort *)
						_ProgramState := BACnetProgramState_halted;
						_ActiveChange := BACnetProgramRequest_ready;
						_ReasonForHalt := BACnetProgramError_other;
					ELSIF stDoneFlags.bUnload THEN
						(* DONE *)
						_ActiveChange := BACnetProgramRequest_ready;
						_ProgramState := BACnetProgramState_idle;
					ELSIF (NOT _bLockedForChange) THEN
						CASE _ProgramChange OF
							BACnetProgramRequest_load,
							BACnetProgramRequest_run,
							BACnetProgramRequest_halt,
							BACnetProgramRequest_restart,
							BACnetProgramRequest_unload:
								(* acknowledge without execution *)
								_SetProgramReadyState	:= TRUE;
						END_CASE
					END_IF
				END_IF

		END_CASE
	END_IF

	(* check state of "change" request *)
	IF (_ActiveChange <> BACnetProgramRequest_ready) THEN
		(* request is active, lock execution *)
		_bLockedForChange		:= TRUE;
	ELSIF _bLockedForChange AND (NOT _SetProgramReadyState) THEN
		(* change finished, tell the stack done *)
		_SetProgramReadyState	:= TRUE;
		_bTriggerSetup			:= FALSE;
	ELSIF (_ProgramChange = BACnetProgramRequest_ready) THEN
		(* wait on new requests *)
		_SetProgramReadyState	:= FALSE;
		_bLockedForChange		:= FALSE;
		_bTriggerSetup			:= FALSE;
	ELSE
		(* new request *)
		_bTriggerSetup			:= FALSE;
	END_IF

	(* external requests *)
	stRequestFlags.bLoad			:= (_ProgramState = BACnetProgramState_loading) AND (NOT _bLockedForChange);
	stRequestFlags.bSetup			:=	(		(_ActiveChange = BACnetProgramRequest_run)
										OR	(_ActiveChange = BACnetProgramRequest_restart)
									)
								AND	_bTriggerSetup;
	stRequestFlags.bRun			:= (_ActiveChange = BACnetProgramRequest_run) AND (NOT _bTriggerSetup);
	stRequestFlags.bHalt			:= _ActiveChange = BACnetProgramRequest_halt;
	stRequestFlags.bUnload		:=	(_ActiveChange = BACnetProgramRequest_unload)
								OR	(		(_ProgramState = BACnetProgramState_unloading)
										AND	(NOT _bLockedForChange)
									);

	(* active status flags *)
	stActiveStateFlags.bIdle		:= _ProgramState = BACnetProgramState_idle;
	stActiveStateFlags.bLoading		:= _ProgramState = BACnetProgramState_loading;
	stActiveStateFlags.bRunning		:= _ProgramState = BACnetProgramState_running;
	stActiveStateFlags.bWaiting		:= _ProgramState = BACnetProgramState_waiting;
	stActiveStateFlags.bHalted		:= _ProgramState = BACnetProgramState_halted;
	stActiveStateFlags.bUnloading	:= _ProgramState = BACnetProgramState_unloading;
ELSE
	(* server device not ready, reset local ready also *)
	bReady := FALSE;
	nErrorId := nERR_OPERATIONAL;
END_IF
(* set error flag *)
bError := (nErrorId <> nERR_NO_ERROR);
END_FUNCTION_BLOCK

(* POU FB_BACnet_ReadProp, ST *)
FUNCTION_BLOCK FB_BACnet_ReadProp
VAR_INPUT
	BACnetDevicePort	: UINT := 16#FFFF;
	bExecute			: BOOL;
	sNetId				: T_AmsNetId;
	ObjectType			: E_BACNETOBJECTTYPE;
	PropertyID			: E_BACNETPROPERTYIDENTIFIER;
	DataType			: E_BACNETDATATYPES;
	ObjectInstance		: DINT;
	ptrValue			: POINTER TO BYTE;
	nLenValue			: UDINT; (* byte size of value (SIZEOF) *)
END_VAR
VAR_OUTPUT
	bDone				: BOOL;
	bBusy				: BOOL;
	bError				: BOOL;
	nErrID				: UDINT;
	nProcessedLen		: UDINT; (* the received data length (can be different to given length) *)
END_VAR
VAR
	_Read				: FW_AdsRead;
	_rtrigStart			: R_TRIG;
	_len_data			: UDINT;
END_VAR
(* catch the start flag *)
	_rtrigStart(Clk:=bExecute);

(* prepare *)
	IF _rtrigStart.Q AND (NOT bBusy) THEN
		_Read(bExecute := FALSE);
		bDone := FALSE;
		bBusy := TRUE;
		bError := FALSE;
		nErrId := 0;
		nProcessedLen := 0;
		(* in default, take the user given length *)
		_len_data := nLenValue;
		(* set index group for read property access *)
		_Read.nIdxGrp := 16#80000000 + INT_TO_UDINT(PropertyID);
		(* handle special data type things *)
		CASE DataType OF
			BACnetDataType_Null 				: _len_data := 0; (* set length to zero *)
			BACnetDataType_Bool 				: _len_data := _len_data; (* 1 *)
			BACnetDataType_CharacterStringExt	: _len_data := _len_data; (* 2 *)
			BACnetDataType_UnsignedInteger 		: _len_data := _len_data; (* 4 *)
			BACnetDataType_SignedInteger 		: _len_data := _len_data; (* 4 *)
			BACnetDataType_Real 				: _len_data := _len_data; (* 4 *)
			BACnetDataType_Double 				: _len_data := _len_data; (* 8 *)
			BACnetDataType_OctetString 			: _len_data := _len_data; (* 8 *)
			BACnetDataType_Enumerated 			: _len_data := _len_data; (* 8 *)
			BACnetDataType_LimitEnable			: _len_data := _len_data; (* 4 *)
			BACnetDataType_BitString 			: _len_data := _len_data; (* 11 *)
			BACnetDataType_LogRecordList:
				_len_data := _len_data; (* n *)
				_Read.nIdxGrp := _Read.nIdxGrp + 16#03800000; (* read range *)
		END_CASE;
	END_IF



(* execute *)
	IF bBusy THEN
		_Read(
			sNetId		:= sNetId,
			nPort		:= BACnetDevicePort,
			nIdxGrp		:= , (* see above *)
			nIdxOffs	:= F_BACnet_GetObjId(ObjectType, ObjectInstance),
			cbReadLen	:= _len_data,
			pReadBuff	:= ptrValue,
			bExecute	:= TRUE,
			tTimeout	:= tBACnet_ADSTimeOut,
			bBusy		=> ,
			bError		=> ,
			nErrId		=> ,
			cbRead		=> );
		IF (NOT _Read.bBusy) THEN
			IF _Read.bError THEN
				nErrID := _Read.nErrId;
				bError := TRUE;
				nProcessedLen := 0;
			ELSE
				nProcessedLen := _Read.cbRead;
			END_IF
			_Read(bExecute := FALSE);
			bBusy := FALSE;
			bDone := NOT bError;
		END_IF;
	END_IF
END_FUNCTION_BLOCK

(* POU FB_BACnet_RemoteAccumulator, ST *)
FUNCTION_BLOCK FB_BACnet_RemoteAccumulator
VAR_IN_OUT
	RemoteDevice		: FB_BACnet_RemoteDevice;
END_VAR
VAR_OUTPUT
	bReady				: BOOL;
	nPresentValue		: UDINT;
	bOverridden			: BOOL;
	bOutOfService		: BOOL;
	bFault				: BOOL;
	bInAlarm			: BOOL;
	bError				: BOOL;
	nErrorId			: UINT;
END_VAR
VAR CONSTANT
	nERR_NO_ERROR		: UINT := 0;
	nERR_REMOTE_DEVICE	: UINT := 1;
	nERR_WRONG_MAPPING	: UINT := 2;
	nERR_OPERATIONAL	: UINT := 3;
END_VAR
VAR
	_PresentValue AT%I*:UDINT;		(* ~(BACnet_PresentValue				:		: )
										(BACnet_ObjectType					: ACC	: )
										(BACnet_RemoteCycletimeRead			: 1000	: )
										(BACnet_RemoteFlagsRead				: 1		: )
										(BACnet_RemoteResubscriptionInterval: 240	: )
                                		(BACnet_RemoteCycleTimeWrite   		: 1000	: )
                                		(BACnet_RemoteFlagsWrite       		: 1		: )	*)
	_StatusFlags AT%I*:WORD;		(* ~(BACnet_StatusFlags					:		: )	*)
	_StatusFlagsBits : ST_BACnet_StatusFlags;

	_nUpdateCount : UDINT := 0;
END_VAR
(* update client device *)
IF RemoteDevice._nUpdateCount = _nUpdateCount THEN
	RemoteDevice();
END_IF
(* remind current number of update counter *)
_nUpdateCount := RemoteDevice._nUpdateCount;

IF _StatusFlags < 4 THEN
	(* mapping seems to be wrong (bit string for status flags must be 4 in minimum) *)
	nErrorId := nERR_WRONG_MAPPING;

ELSIF RemoteDevice.bOperational THEN
	(* clear error flag *)
	nErrorId := nERR_NO_ERROR;
	bReady := TRUE;
	(* copy present value *)
	nPresentValue := _PresentValue;

	(* build bit states *)
	_StatusFlagsBits := F_BACnet_StatusFlags(_StatusFlags);

	(* copy states to output *)
	bOverridden := _StatusFlagsBits.overridden;
	bOutOfService := _StatusFlagsBits.out_of_service;
	bFault := _StatusFlagsBits.fault;
	bInAlarm := _StatusFlagsBits.in_alarm;
ELSE
	bReady := FALSE;
	(* and set error ID *)
	nErrorId := nERR_OPERATIONAL;
END_IF

(* set error flag *)
bError := (nErrorId <> nERR_NO_ERROR);
END_FUNCTION_BLOCK

(* POU FB_BACnet_RemoteDevice, ST *)
FUNCTION_BLOCK FB_BACnet_RemoteDevice
VAR_INPUT
	bReset				: BOOL;
	bAutoReset			: BOOL;
	bDisableWOC			: BOOL;
	bReSubscribeCOV		: BOOL;
	bAutoReSubscribe	: BOOL;
END_VAR
VAR_OUTPUT
	eSystemStatus		: E_BACNETDEVICESTATUS;
	bEthLinkOk			: BOOL;
	bGatewayOk			: BOOL;
	sAmsNetId			: T_AmsNetId;
	bEnabledWOC			: BOOL;
	bOperational		: BOOL;
	bConnecting			: BOOL;
	bFirstCycle			: BOOL;
	bError				: BOOL;
	nErrorId			: UINT;
	bClientTimeout		: BOOL;
	bServiceFailed		: BOOL;
	nTimeoutCnt			: UDINT;
	nServiceFailCnt		: UDINT;
END_VAR
VAR CONSTANT
	nERR_NO_ERROR		: UINT := 0;
(* errors without reset 1..19 *)
	nERR_NO_VALID_NET_ID	: UINT := 1;
	nERR_NO_ETH_LINK		: UINT := 3;
	nERR_NO_GATEWAY			: UINT := 4;

(* errors with reset 20.. *)
	nERR_CLIENT_TIMEOUT	: UINT := 20;
	nERR_CLIENT_SERVICE	: UINT := 21;
END_VAR
VAR
	_SystemStatus AT%I*	: E_BACNETDEVICESTATUS;
									(* ~(BACnet_SystemStatus 				: 		: )
										(BACnet_ObjectType					: DEV	: )
				                        (BACnet_RemoteCycletimeRead 		: 5000	: ) polling each 5 seconds
										(BACnet_RemoteFlagsRead        		: 2     : ) 2 = polling, so the object detects if the client is unreachable!
	                                   	(BACnet_RemoteResubscriptionInterval: 240 	: )
	                            		(BACnet_RemoteCycleTimeWrite   		: 1000	: )
                            			(BACnet_RemoteFlagsWrite       		: 1		: )  
		   							*)
	_ClientStatus AT%I*	:WORD;		(* ~(BACnet_ClientStatus				:		: )	*)
	_ObjIdentifier AT%I* : DWORD;	(* ~(BACnet_ObjectIdentifier			:		: LINK ) *)
	_ClientControl AT%Q*:WORD;		(* ~(BACnet_ClientControl				:		: ) *)
	_rtrigReset			: R_TRIG;
	_rtrigOperational	: R_TRIG;
	_rtrigResubscribe	: R_TRIG;
	_rtrigTimeoutCnt	: R_TRIG;
	_rtrigServiceFailCnt: R_TRIG;
	_bReqResubscribe	: BOOL;
	_bComplete			: BOOL;
	_tofTimeoutLeft		: TOF;
	_tofServiceErrLeft	: TOF;
	_ftrigTimeoutLeft	: F_TRIG;

	_bHasStarted		: BOOL := TRUE;
	_nUpdateCount		: UDINT := 0;
	_nUpdateCountAdp 	: UDINT := 0;
	_BACnetAdapter		: POINTER TO FB_BACnet_Adapter;
END_VAR
(* check pointer to bacnet adapter instance *)
IF pBACnet_Adapter > 0 THEN
	_BACnetAdapter := pBACnet_Adapter;
ELSE
	_BACnetAdapter := ADR(fbBACnet_Adapter);
END_IF

(* update server device *)
IF _BACnetAdapter^._nUpdateCount = _nUpdateCountAdp THEN
	_BACnetAdapter^();
END_IF
(* remind current number of update counter *)
_nUpdateCountAdp := _BACnetAdapter^._nUpdateCount;

(* convert SystemStatus to enumeration *)
eSystemStatus := _SystemStatus;
(* reset trigger *)
_rtrigReset(CLK:= bReset, Q=> );
(* reset error ID and flag *)
IF (nErrorId < 20) OR _rtrigReset.Q OR bAutoReset THEN
	bError := FALSE;
	nErrorId := nERR_NO_ERROR;
END_IF
IF _rtrigReset.Q OR (NOT _bComplete) OR bAutoReset THEN
	_ClientControl.0 := _ClientStatus.0;
	_ClientControl.1 := _ClientStatus.1;
END_IF

(* read NetId and convert to string *)
sAmsNetId := _BACnetAdapter^.sAmsNetId;
(* check if it plausible *)
IF sAmsNetId = '' THEN
	(* NetId not OK, return with error *)
	bError := TRUE;
	nErrorId := nERR_NO_VALID_NET_ID;
ELSIF (NOT _BACnetAdapter^.bEthLinkOk) THEN
	(* ethernet link missing *)
	bError := TRUE;
	nErrorId := nERR_NO_ETH_LINK;
ELSIF (NOT _BACnetAdapter^.bGatewayOk) THEN
	(* gateway missing *)
	bError := TRUE;
	nErrorId := nERR_NO_GATEWAY;
END_IF

(* check for client errors *)
IF _ClientStatus.0 AND _bComplete THEN
	nErrorId := nERR_CLIENT_TIMEOUT;
	bError := TRUE;
ELSIF _ClientStatus.1 AND _bComplete THEN
	nErrorId := nERR_CLIENT_SERVICE;
	bError := TRUE;
ELSE
	(* reset both acknowledge flags *)
	_ClientControl.0 := FALSE;
	_ClientControl.1 := FALSE;
END_IF

(* summerize timeout errors *)
_rtrigTimeoutCnt(CLK:= _ClientStatus.0, Q=> );
_tofTimeoutLeft(
	IN:= (_rtrigTimeoutCnt.Q AND _bComplete),
	PT:= T#10s,
	Q=> bClientTimeout,
	ET=> );
IF _tofTimeoutLeft.IN THEN
	nTimeoutCnt := nTimeoutCnt + 1;
END_IF
_ftrigTimeoutLeft(CLK:= _tofTimeoutLeft.Q, Q=> );

(* summerize service errors *)
_rtrigServiceFailCnt(CLK:= _ClientStatus.1, Q=> );
_tofServiceErrLeft(
	IN:= (_rtrigServiceFailCnt.Q AND _bComplete),
	PT:= T#10s,
	Q=> bServiceFailed,
	ET=> );
IF _tofServiceErrLeft.IN THEN
	nServiceFailCnt := nServiceFailCnt + 1;
END_IF

(* controls *)
_ClientControl.2 := bDisableWOC;
_ClientControl.3 := _bReqResubscribe;

(* states *)
bEthLinkOk := _BACnetAdapter^.bEthLinkOk;
bGatewayOk := _BACnetAdapter^.bGatewayOk;

bEnabledWOC := (NOT _ClientStatus.2);
bConnecting := (SHR((_ClientStatus AND 16#FF00), 8) < 4);
_bComplete :=		(NOT bConnecting)
				AND	(_SystemStatus = 0)
				AND	_BACnetAdapter^.bEthLinkOk;
bOperational :=		_bComplete
				AND ((NOT _ClientStatus.0) OR bAutoReset);

(* Resubscribe COV *)
_rtrigOperational(CLK:= bOperational, Q=> );
_rtrigResubscribe(CLK:= bReSubscribeCOV, Q=> );
IF		(		(		(		_rtrigOperational.Q
							OR (_ftrigTimeoutLeft.Q AND bAutoReset)
						)
					AND	bAutoReSubscribe
				)
			OR	_rtrigResubscribe.Q
		)
	AND	(NOT _bReqResubscribe)
THEN
	(* operation mode reached or resubscription was externally triggered, start resubcription *)
	_bReqResubscribe	:= TRUE;
ELSIF (NOT bOperational) THEN
	(* not operational *)
	_bReqResubscribe	:= FALSE;
ELSE
	IF _bReqResubscribe AND _ClientStatus.3 THEN
		(* resubscription triggered *)
		_bReqResubscribe := FALSE;
	END_IF
END_IF

(* update counter *)
IF (_nUpdateCount = 0) AND _bHasStarted THEN
	bFirstCycle := TRUE;
	_bHasStarted := FALSE;
ELSE
	bFirstCycle := FALSE;
END_IF
_nUpdateCount := _nUpdateCount +1;
END_FUNCTION_BLOCK

(* POU FB_BACnet_RemoteAccumulator_EX, ST *)
FUNCTION_BLOCK FB_BACnet_RemoteAccumulator_EX
VAR_IN_OUT
	RemoteDevice		: FB_BACnet_RemoteDevice;
END_VAR
VAR_OUTPUT
	bReady				: BOOL;
	nPresentValue		: UDINT;
	bOverridden			: BOOL;
	bOutOfService		: BOOL;
	bFault				: BOOL;
	bInAlarm			: BOOL;
	bOverRange			: BOOL;
	bUnderRange			: BOOL;
	bOpenLoop			: BOOL;
	bShortedLoop		: BOOL;
	bOtherFault			: BOOL;
	bError				: BOOL;
	nErrorId			: UINT;
END_VAR
VAR CONSTANT
	nERR_NO_ERROR		: UINT := 0;
	nERR_REMOTE_DEVICE	: UINT := 1;
	nERR_WRONG_MAPPING	: UINT := 2;
	nERR_OPERATIONAL	: UINT := 3;
END_VAR
VAR
	_PresentValue AT%I*:UDINT;		(* ~(BACnet_PresentValue				:		: )
										(BACnet_ObjectType					: ACC	: )
										(BACnet_RemoteCycletimeRead			: 1000	: )
										(BACnet_RemoteFlagsRead				: 1		: )
										(BACnet_RemoteResubscriptionInterval: 240	: )
                                		(BACnet_RemoteCycleTimeWrite   		: 1000	: )
                                		(BACnet_RemoteFlagsWrite       		: 1		: )	*)
	_StatusFlags AT%I*:WORD;		(* ~(BACnet_StatusFlags					:		: )	*)
	_Reliability AT%I*:WORD;		(* ~(BACnet_Reliability					:		: )	*)
	_StatusFlagsBits : ST_BACnet_StatusFlags;

	_nUpdateCount : UDINT := 0;
END_VAR
(* update client device *)
IF RemoteDevice._nUpdateCount = _nUpdateCount THEN
	RemoteDevice();
END_IF
(* remind current number of update counter *)
_nUpdateCount := RemoteDevice._nUpdateCount;

IF _StatusFlags < 4 THEN
	(* mapping seems to be wrong (bit string for status flags must be 4 in minimum) *)
	nErrorId := nERR_WRONG_MAPPING;

ELSIF RemoteDevice.bOperational THEN
	(* clear error flag *)
	nErrorId := nERR_NO_ERROR;
	bReady := TRUE;
	(* copy present value *)
	nPresentValue := _PresentValue;

	(* build bit states *)
	_StatusFlagsBits := F_BACnet_StatusFlags(_StatusFlags);

	(* copy states to output *)
	bOverridden := _StatusFlagsBits.overridden;
	bOutOfService := _StatusFlagsBits.out_of_service;
	bFault := _StatusFlagsBits.fault;
	bInAlarm := _StatusFlagsBits.in_alarm;
	bOverRange := (_Reliability = BACnetReliability_over_range);
	bUnderRange := (_Reliability = BACnetReliability_under_range);
	bOpenLoop := (_Reliability = BACnetReliability_open_loop);
	bShortedLoop := (_Reliability = BACnetReliability_shorted_loop);
	bOtherFault := (_Reliability = BACnetReliability_unreliable_other);
ELSE
	bReady := FALSE;
	(* and set error ID *)
	nErrorId := nERR_OPERATIONAL;
END_IF

(* set error flag *)
bError := (nErrorId <> nERR_NO_ERROR);
END_FUNCTION_BLOCK

(* POU FB_BACnet_RemoteAnalogInput, ST *)
FUNCTION_BLOCK FB_BACnet_RemoteAnalogInput
VAR_IN_OUT
	RemoteDevice			: FB_BACnet_RemoteDevice;
END_VAR
VAR_OUTPUT
	bReady				: BOOL;
	fPresentValue		: REAL;
	bOverridden			: BOOL;
	bOutOfService		: BOOL;
	bFault				: BOOL;
	bInAlarm			: BOOL;
	bError				: BOOL;
	nErrorId			: UINT;
END_VAR
VAR CONSTANT
	nERR_NO_ERROR		: UINT := 0;
	nERR_REMOTE_DEVICE	: UINT := 1;
	nERR_WRONG_MAPPING	: UINT := 2;
	nERR_OPERATIONAL	: UINT := 3;
END_VAR
VAR
	_PresentValue AT%I*: REAL; 			(* ~(BACnet_PresentValue 				:		: )
								   			(BACnet_ObjectType 					: AI	: )
											(BACnet_RemoteCycletimeRead 		: 1000	: )
											(BACnet_RemoteFlagsRead        		: 1		: )
											(BACnet_RemoteResubscriptionInterval: 240	: )
	                                		(BACnet_RemoteCycleTimeWrite   		: 1000	: )
	                                		(BACnet_RemoteFlagsWrite       		: 1		: )	*)
	_StatusFlags AT%I*: WORD; 			(* ~(BACnet_StatusFlags 				:		: )	*)
	_StatusFlagsBits : ST_BACnet_StatusFlags;

	_nUpdateCount : UDINT := 0;
END_VAR
(* update client device *)
IF RemoteDevice._nUpdateCount = _nUpdateCount THEN
	RemoteDevice();
END_IF
(* remind current number of update counter *)
_nUpdateCount := RemoteDevice._nUpdateCount;

IF _StatusFlags < 4 THEN
	(* mapping seems to be wrong (bit string for status flags must be 4 in minimum) *)
	nErrorId := nERR_WRONG_MAPPING;

ELSIF RemoteDevice.bOperational THEN
	(* clear error flag *)
	nErrorId := nERR_NO_ERROR;
	(* ready state *)
	bReady := TRUE;

	(* present value *)
	fPresentValue := _PresentValue;

	(* build bit states *)
	_StatusFlagsBits := F_BACnet_StatusFlags(_StatusFlags);

	(* copy states to output *)
	bOverridden := _StatusFlagsBits.overridden;
	bOutOfService := _StatusFlagsBits.out_of_service;
	bFault := _StatusFlagsBits.fault;
	bInAlarm := _StatusFlagsBits.in_alarm;
ELSE
	(* server device not ready, reset local ready also *)
	bReady := FALSE;
	(* and set error ID *)
	nErrorId := nERR_OPERATIONAL;
END_IF

(* set error flag *)
bError := (nErrorId <> nERR_NO_ERROR);
END_FUNCTION_BLOCK

(* POU FB_BACnet_RemoteAnalogInput_EX, ST *)
FUNCTION_BLOCK FB_BACnet_RemoteAnalogInput_EX
VAR_IN_OUT
	RemoteDevice			: FB_BACnet_RemoteDevice;
END_VAR
VAR_OUTPUT
	bReady				: BOOL;
	fPresentValue		: REAL;
	bOverridden			: BOOL;
	bOutOfService		: BOOL;
	bFault				: BOOL;
	bInAlarm			: BOOL;
	bOverRange			: BOOL;
	bUnderRange			: BOOL;
	bNoSensor			: BOOL;
	bOpenLoop			: BOOL;
	bShortedLoop		: BOOL;
	bOtherFault			: BOOL;
	eEventState			: E_BACNETEVENTSTATE;
	bError				: BOOL;
	nErrorId			: UINT;
END_VAR
VAR CONSTANT
	nERR_NO_ERROR		: UINT := 0;
	nERR_REMOTE_DEVICE	: UINT := 1;
	nERR_WRONG_MAPPING	: UINT := 2;
	nERR_OPERATIONAL	: UINT := 3;
END_VAR
VAR
	_PresentValue AT%I*: REAL; 			(* ~(BACnet_PresentValue 				:		: )
								   			(BACnet_ObjectType 					: AI	: )
											(BACnet_RemoteCycletimeRead 		: 1000	: )
											(BACnet_RemoteFlagsRead        		: 1		: )
											(BACnet_RemoteResubscriptionInterval: 240	: )
	                                		(BACnet_RemoteCycleTimeWrite   		: 1000	: )
	                                		(BACnet_RemoteFlagsWrite       		: 1		: )	*)
	_StatusFlags AT%I*: WORD; 			(* ~(BACnet_StatusFlags 				:		: )	*)
	_StatusFlagsBits : ST_BACnet_StatusFlags;
	_Reliability AT%I*: WORD; 			(* ~(BACnet_Reliability 				:		: )	*)
	_EventState AT%I*: WORD;			(* ~(BACnet_EventState					:		: )	*)

	_nUpdateCount : UDINT := 0;
END_VAR
(* update client device *)
IF RemoteDevice._nUpdateCount = _nUpdateCount THEN
	RemoteDevice();
END_IF
(* remind current number of update counter *)
_nUpdateCount := RemoteDevice._nUpdateCount;

IF _StatusFlags < 4 THEN
	(* mapping seems to be wrong (bit string for status flags must be 4 in minimum) *)
	nErrorId := nERR_WRONG_MAPPING;

ELSIF RemoteDevice.bOperational THEN
	(* clear error flag *)
	nErrorId := nERR_NO_ERROR;
	(* ready state *)
	bReady := TRUE;

	(* present value *)
	fPresentValue := _PresentValue;

	(* build bit states *)
	_StatusFlagsBits := F_BACnet_StatusFlags(_StatusFlags);

	(* copy states to output *)
	bOverridden := _StatusFlagsBits.overridden;
	bOutOfService := _StatusFlagsBits.out_of_service;
	bFault := _StatusFlagsBits.fault;
	bInAlarm := _StatusFlagsBits.in_alarm;
	bOverRange := (_Reliability = BACnetReliability_over_range);
	bUnderRange := (_Reliability = BACnetReliability_under_range);
	bNoSensor := (_Reliability = BACnetReliability_no_sensor);
	bOpenLoop := (_Reliability = BACnetReliability_open_loop);
	bShortedLoop := (_Reliability = BACnetReliability_shorted_loop);
	bOtherFault := (_Reliability = BACnetReliability_unreliable_other);
	eEventState := _EventState;
ELSE
	(* server device not ready, reset local ready also *)
	bReady := FALSE;
	(* and set error ID *)
	nErrorId := nERR_OPERATIONAL;
END_IF

(* set error flag *)
bError := (nErrorId <> nERR_NO_ERROR);
END_FUNCTION_BLOCK

(* POU FB_BACnet_RemoteAnalogOutput, ST *)
FUNCTION_BLOCK FB_BACnet_RemoteAnalogOutput
VAR_INPUT
	bEnablePV		: BOOL; (* enable present value with priority x in priority array, FALSE = priority x disable *)
	fPV		: REAL; (* decimal number for priority x, when input bEnablePV is TRUE *)
END_VAR
VAR_IN_OUT
	RemoteDevice	: FB_BACnet_RemoteDevice;
END_VAR
VAR_OUTPUT
	bReady				: BOOL;
	fPresentValue		: REAL;
	bOverridden			: BOOL;
	bOutOfService		: BOOL;
	bFault				: BOOL;
	bInAlarm			: BOOL;
	bError				: BOOL;
	nErrorId			: UINT;
END_VAR
VAR CONSTANT
	nERR_NO_ERROR		: UINT := 0;
	nERR_REMOTE_DEVICE	: UINT := 1;
	nERR_WRONG_MAPPING	: UINT := 2;
	nERR_OPERATIONAL	: UINT := 3;
END_VAR
VAR
	_PresentValue AT%I*: REAL; 			(* ~(BACnet_PresentValue 				:		: )
								   			(BACnet_ObjectType 					: AO	: )
											(BACnet_RemoteCycletimeRead 		: 1000	: )
											(BACnet_RemoteFlagsRead        		: 1		: )
											(BACnet_RemoteResubscriptionInterval: 240	: )
	                                		(BACnet_RemoteCycleTimeWrite   		: 1000	: )
	                                		(BACnet_RemoteFlagsWrite       		: 1		: )	*)
    _PresentValue_Priority12 AT%Q*: REAL;(* ~(BACnet_PresentValue_Priority12		:		: )	*)
	_StatusFlags AT%I*: WORD; 			(* ~(BACnet_StatusFlags 				:		: )	*)
	_StatusFlagsBits : ST_BACnet_StatusFlags;

	_nUpdateCount : UDINT := 0;
END_VAR
(* update client device *)
IF RemoteDevice._nUpdateCount = _nUpdateCount THEN
	RemoteDevice();
END_IF
(* remind current number of update counter *)
_nUpdateCount := RemoteDevice._nUpdateCount;

IF _StatusFlags < 4 THEN
	(* mapping seems to be wrong (bit string for status flags must be 4 in minimum) *)
	nErrorId := nERR_WRONG_MAPPING;

ELSIF RemoteDevice.bOperational THEN
	(* clear error flag *)
	nErrorId := nERR_NO_ERROR;
	(* ready state *)
	bReady := TRUE;

	(* write into priority array *)
	IF bEnablePV THEN
		_PresentValue_Priority12	:= fPV;
	ELSE
		_PresentValue_Priority12	:= F_BACnet_NAN();
	END_IF

	(* present value *)
	fPresentValue := _PresentValue;

	(* build bit states *)
	_StatusFlagsBits := F_BACnet_StatusFlags(_StatusFlags);

	(* copy states to output *)
	bOverridden := _StatusFlagsBits.overridden;
	bOutOfService := _StatusFlagsBits.out_of_service;
	bFault := _StatusFlagsBits.fault;
	bInAlarm := _StatusFlagsBits.in_alarm;
ELSIF RemoteDevice.bFirstCycle THEN
	(* first call of the server device since reboot/reset *)
	bReady := FALSE;
	_PresentValue_Priority12 := F_BACnet_NAN();
ELSE
	(* server device not ready, reset local ready also *)
	bReady := FALSE;
	(* and set error ID *)
	nErrorId := nERR_OPERATIONAL;
END_IF

(* set error flag *)
bError := (nErrorId <> nERR_NO_ERROR);
END_FUNCTION_BLOCK

(* POU FB_BACnet_RemoteAnalogOutput_EX, ST *)
FUNCTION_BLOCK FB_BACnet_RemoteAnalogOutput_EX
VAR_INPUT
	bEnablePV		: BOOL; (* enable present value with priority x in priority array, FALSE = priority x disable *)
	fPV		: REAL; (* decimal number for priority x, when input bEnablePV is TRUE *)
END_VAR
VAR_IN_OUT
	RemoteDevice	: FB_BACnet_RemoteDevice;
END_VAR
VAR_OUTPUT
	bReady				: BOOL;
	fPresentValue		: REAL;
	bOverridden			: BOOL;
	bOutOfService		: BOOL;
	bFault				: BOOL;
	bInAlarm			: BOOL;
	bNoOutput			: BOOL;
	bOpenLoop			: BOOL;
	bShortedLoop		: BOOL;
	bOtherFault			: BOOL;
	eEventState			: E_BACNETEVENTSTATE;
	bError				: BOOL;
	nErrorId			: UINT;
END_VAR
VAR CONSTANT
	nERR_NO_ERROR		: UINT := 0;
	nERR_REMOTE_DEVICE	: UINT := 1;
	nERR_WRONG_MAPPING	: UINT := 2;
	nERR_OPERATIONAL	: UINT := 3;
END_VAR
VAR
	_PresentValue AT%I*: REAL; 			(* ~(BACnet_PresentValue 				:		: )
								   			(BACnet_ObjectType 					: AO	: )
											(BACnet_RemoteCycletimeRead 		: 1000	: )
											(BACnet_RemoteFlagsRead        		: 1		: )
											(BACnet_RemoteResubscriptionInterval: 240	: )
	                                		(BACnet_RemoteCycleTimeWrite   		: 1000	: )
	                                		(BACnet_RemoteFlagsWrite       		: 1		: )	*)
    _PresentValue_Priority12 AT%Q*: REAL;(* ~(BACnet_PresentValue_Priority12		:		: )	*)
	_StatusFlags AT%I*: WORD; 			(* ~(BACnet_StatusFlags 				:		: )	*)
	_StatusFlagsBits : ST_BACnet_StatusFlags;
	_Reliability AT%I*: WORD; 			(* ~(BACnet_Reliability 				:		: )	*)
	_EventState AT%I*: WORD;			(* ~(BACnet_EventState					:		: )	*)

	_nUpdateCount : UDINT := 0;
END_VAR
(* update client device *)
IF RemoteDevice._nUpdateCount = _nUpdateCount THEN
	RemoteDevice();
END_IF
(* remind current number of update counter *)
_nUpdateCount := RemoteDevice._nUpdateCount;

IF _StatusFlags < 4 THEN
	(* mapping seems to be wrong (bit string for status flags must be 4 in minimum) *)
	nErrorId := nERR_WRONG_MAPPING;

ELSIF RemoteDevice.bOperational THEN
	(* clear error flag *)
	nErrorId := nERR_NO_ERROR;
	(* ready state *)
	bReady := TRUE;

	(* write into priority array *)
	IF bEnablePV THEN
		_PresentValue_Priority12	:= fPV;
	ELSE
		_PresentValue_Priority12	:= F_BACnet_NAN();
	END_IF

	(* present value *)
	fPresentValue := _PresentValue;

	(* build bit states *)
	_StatusFlagsBits := F_BACnet_StatusFlags(_StatusFlags);

	(* copy states to output *)
	bOverridden := _StatusFlagsBits.overridden;
	bOutOfService := _StatusFlagsBits.out_of_service;
	bFault := _StatusFlagsBits.fault;
	bInAlarm := _StatusFlagsBits.in_alarm;
	bNoOutput := (_Reliability = BACnetReliability_no_output);
	bOpenLoop := (_Reliability = BACnetReliability_open_loop);
	bShortedLoop := (_Reliability = BACnetReliability_shorted_loop);
	bOtherFault := (_Reliability = BACnetReliability_unreliable_other);
	eEventState := _EventState;
ELSIF RemoteDevice.bFirstCycle THEN
	(* first call of the server device since reboot/reset *)
	bReady := FALSE;
	_PresentValue_Priority12 := F_BACnet_NAN();
ELSE
	(* server device not ready, reset local ready also *)
	bReady := FALSE;
	(* and set error ID *)
	nErrorId := nERR_OPERATIONAL;
END_IF

(* set error flag *)
bError := (nErrorId <> nERR_NO_ERROR);
END_FUNCTION_BLOCK

(* POU FB_BACnet_RemoteAnalogValue, ST *)
FUNCTION_BLOCK FB_BACnet_RemoteAnalogValue
VAR_INPUT
	bEnablePV		: BOOL; (* enable present value with priority x in priority array, FALSE = priority x disable *)
	fPV		: REAL; (* decimal number for priority x, when input bEnablePV is TRUE *)
END_VAR
VAR_IN_OUT
	RemoteDevice	: FB_BACnet_RemoteDevice;
END_VAR
VAR_OUTPUT
	bReady				: BOOL;
	fPresentValue		: REAL;
	bOverridden			: BOOL;
	bOutOfService		: BOOL;
	bFault				: BOOL;
	bInAlarm			: BOOL;
	bError				: BOOL;
	nErrorId			: UINT;
END_VAR
VAR CONSTANT
	nERR_NO_ERROR		: UINT := 0;
	nERR_REMOTE_DEVICE	: UINT := 1;
	nERR_WRONG_MAPPING	: UINT := 2;
	nERR_OPERATIONAL	: UINT := 3;
END_VAR
VAR
	_PresentValue AT%I*: REAL; 			(* ~(BACnet_PresentValue 				:		: )
								   			(BACnet_ObjectType 					: AV	: )
											(BACnet_RemoteCycletimeRead 		: 1000	: )
											(BACnet_RemoteFlagsRead        		: 1		: )
											(BACnet_RemoteResubscriptionInterval: 240	: )
	                                		(BACnet_RemoteCycleTimeWrite   		: 1000	: )
	                                		(BACnet_RemoteFlagsWrite       		: 1		: )	*)
    _PresentValue_Priority12 AT%Q*: REAL;(* ~(BACnet_PresentValue_Priority12		:		: )	*)
	_StatusFlags AT%I*: WORD; 			(* ~(BACnet_StatusFlags 				:		: )	*)
	_StatusFlagsBits : ST_BACnet_StatusFlags;

	_nUpdateCount : UDINT := 0;
END_VAR
(* update client device *)
IF RemoteDevice._nUpdateCount = _nUpdateCount THEN
	RemoteDevice();
END_IF
(* remind current number of update counter *)
_nUpdateCount := RemoteDevice._nUpdateCount;

IF _StatusFlags < 4 THEN
	(* mapping seems to be wrong (bit string for status flags must be 4 in minimum) *)
	nErrorId := nERR_WRONG_MAPPING;

ELSIF RemoteDevice.bOperational THEN
	(* clear error flag *)
	nErrorId := nERR_NO_ERROR;
	(* ready state *)
	bReady := TRUE;

	(* write into priority array *)
	IF bEnablePV THEN
		_PresentValue_Priority12	:= fPV;
	ELSE
		_PresentValue_Priority12	:= F_BACnet_NAN();
	END_IF

	(* present value *)
	fPresentValue := _PresentValue;

	(* build bit states *)
	_StatusFlagsBits := F_BACnet_StatusFlags(_StatusFlags);

	(* copy states to output *)
	bOverridden := _StatusFlagsBits.overridden;
	bOutOfService := _StatusFlagsBits.out_of_service;
	bFault := _StatusFlagsBits.fault;
	bInAlarm := _StatusFlagsBits.in_alarm;
ELSIF RemoteDevice.bFirstCycle THEN
	(* first call of the server device since reboot/reset *)
	bReady := FALSE;
	_PresentValue_Priority12 := F_BACnet_NAN();
ELSE
	(* server device not ready, reset local ready also *)
	bReady := FALSE;
	(* and set error ID *)
	nErrorId := nERR_OPERATIONAL;
END_IF

(* set error flag *)
bError := (nErrorId <> nERR_NO_ERROR);
END_FUNCTION_BLOCK

